C03563=1009.631,342.526,-157.819,170.244,53.143,160.444
C03564=1009.638,342.773,-157.854,170.253,53.138,160.444
C03565=1009.644,343.021,-157.889,170.261,53.133,160.445
C03566=1009.650,343.269,-157.924,170.269,53.128,160.445
C03567=1009.657,343.516,-157.959,170.277,53.124,160.446
C03568=1009.664,343.764,-157.994,170.285,53.119,160.447
C03569=1009.671,344.011,-158.030,170.294,53.114,160.447
C03570=1009.677,344.258,-158.064,170.303,53.109,160.448
C03571=1009.683,344.506,-158.100,170.311,53.104,160.448
C03572=1009.689,344.753,-158.135,170.319,53.099,160.449
C03573=1009.696,345.000,-158.170,170.327,53.095,160.450
C03574=1009.703,345.248,-158.205,170.335,53.090,160.450
C03575=1009.709,345.496,-158.241,170.344,53.085,160.450
C03576=1009.716,345.743,-158.276,170.352,53.081,160.451
C03577=1009.723,345.990,-158.311,170.360,53.076,160.452
C03578=1009.729,346.238,-158.347,170.368,53.071,160.452
C03579=1009.735,346.485,-158.382,170.376,53.067,160.453
C03580=1009.741,346.733,-158.418,170.385,53.062,160.453
C03581=1009.748,346.980,-158.453,170.394,53.057,160.454
C03582=1009.755,347.227,-158.490,170.402,53.052,160.454
C03583=1009.761,347.475,-158.525,170.411,53.048,160.455
C03584=1009.767,347.722,-158.561,170.419,53.043,160.456
C03585=1009.775,347.970,-158.597,170.427,53.039,160.456
C03586=1009.782,348.217,-158.632,170.435,53.034,160.457
C03587=1009.788,348.465,-158.668,170.444,53.030,160.458
C03588=1009.795,348.711,-158.703,170.452,53.025,160.458
C03589=1009.801,348.959,-158.739,170.462,53.020,160.459
C03590=1009.808,349.206,-158.775,170.470,53.016,160.459
C03591=1009.814,349.454,-158.811,170.478,53.011,160.460
C03592=1009.822,349.701,-158.847,170.486,53.006,160.461
C03593=1009.828,349.949,-158.883,170.495,53.002,160.461
C03594=1009.835,350.195,-158.919,170.503,52.998,160.462
C03595=1009.841,350.442,-158.955,170.512,52.993,160.463
C03596=1009.848,350.691,-158.991,170.521,52.989,160.463
C03597=1009.855,350.938,-159.027,170.530,52.984,160.464
C03598=1009.862,351.185,-159.062,170.538,52.979,160.465
C03599=1009.869,351.433,-159.099,170.546,52.975,160.465
C03600=1009.876,351.679,-159.135,170.555,52.971,160.466
C03601=1009.882,351.927,-159.171,170.564,52.966,160.467
C03602=1009.889,352.175,-159.207,170.572,52.962,160.467
C03603=1009.896,352.422,-159.243,170.581,52.957,160.468
C03604=1009.903,352.668,-159.279,170.590,52.953,160.469
C03605=1009.910,352.916,-159.316,170.598,52.949,160.469
C03606=1009.916,353.163,-159.352,170.608,52.944,160.470
C03607=1009.922,353.410,-159.389,170.616,52.940,160.471
C03608=1009.930,353.658,-159.425,170.624,52.935,160.471
C03609=1009.936,353.907,-159.462,170.633,52.931,160.472
C03610=1009.944,354.156,-159.498,170.642,52.927,160.473
C03611=1009.950,354.406,-159.536,170.651,52.922,160.474
C03612=1009.957,354.655,-159.572,170.659,52.918,160.474
C03613=1009.964,354.902,-159.609,170.669,52.914,160.475
C03614=1009.971,355.149,-159.645,170.678,52.909,160.476
C03615=1009.978,355.397,-159.681,170.686,52.905,160.477
C03616=1009.985,355.643,-159.719,170.695,52.901,160.477
C03617=1009.993,355.891,-159.755,170.704,52.896,160.478
C03618=1010.000,356.139,-159.792,170.713,52.893,160.479
C03619=1010.006,356.386,-159.828,170.722,52.889,160.480
C03620=1010.013,356.633,-159.866,170.731,52.884,160.481
C03621=1010.020,356.880,-159.901,170.740,52.880,160.481
C03622=1010.027,357.127,-159.938,170.748,52.876,160.482
C03623=1010.034,357.374,-159.976,170.757,52.872,160.483
C03624=1010.041,357.622,-160.012,170.767,52.867,160.484
C03625=1010.049,357.868,-160.049,170.775,52.863,160.485
C03626=1010.056,358.116,-160.086,170.784,52.859,160.485
C03627=1010.062,358.363,-160.123,170.794,52.855,160.486
C03628=1010.070,358.610,-160.161,170.803,52.851,160.487
C03629=1010.077,358.857,-160.197,170.811,52.847,160.488
C03630=1010.084,359.105,-160.235,170.821,52.843,160.489
C03631=1010.090,359.351,-160.272,170.830,52.838,160.489
C03632=1010.098,359.598,-160.310,170.839,52.835,160.490
C03633=1010.105,359.846,-160.347,170.848,52.830,160.491
C03634=1010.112,360.093,-160.384,170.857,52.827,160.492
C03635=1010.119,360.340,-160.422,170.866,52.823,160.493
C03636=1010.126,360.587,-160.459,170.876,52.819,160.494
C03637=1010.133,360.834,-160.496,170.884,52.814,160.495
C03638=1010.140,361.081,-160.534,170.893,52.811,160.495
C03639=1010.147,361.328,-160.571,170.903,52.806,160.496
C03640=1010.155,361.575,-160.609,170.912,52.803,160.497
C03641=1010.162,361.822,-160.646,170.922,52.799,160.498
C03642=1010.169,362.069,-160.684,170.930,52.795,160.499
C03643=1010.176,362.317,-160.721,170.939,52.791,160.500
C03644=1010.184,362.564,-160.759,170.949,52.787,160.501
C03645=1010.191,362.811,-160.796,170.958,52.783,160.502
C03646=1010.198,363.058,-160.834,170.968,52.779,160.503
C03647=1010.205,363.305,-160.872,170.977,52.775,160.504
C03648=1010.213,363.552,-160.910,170.987,52.771,160.505
C03649=1010.220,363.799,-160.947,170.995,52.767,160.505
C03650=1010.227,364.046,-160.985,171.005,52.763,160.506
C03651=1010.235,364.293,-161.022,171.014,52.760,160.507
C03652=1010.242,364.539,-161.061,171.023,52.756,160.508
C03653=1010.250,364.787,-161.098,171.033,52.752,160.509
C03654=1010.257,365.034,-161.136,171.042,52.749,160.510
C03655=1010.265,365.281,-161.174,171.052,52.745,160.511
C03656=1010.272,365.528,-161.212,171.061,52.741,160.512
C03657=1009.942,363.417,-161.243,170.962,52.829,160.514
C03658=1009.935,363.169,-161.206,170.952,52.833,160.513
C03659=1009.928,362.922,-161.168,170.943,52.836,160.512
C03660=1009.920,362.675,-161.131,170.934,52.840,160.511
C03661=1009.913,362.428,-161.093,170.924,52.844,160.510
C03662=1009.906,362.181,-161.056,170.915,52.848,160.509
C03663=1009.899,361.934,-161.018,170.905,52.852,160.508
C03664=1009.891,361.687,-160.981,170.897,52.856,160.508
C03665=1009.884,361.439,-160.943,170.887,52.860,160.507
C03666=1009.877,361.192,-160.906,170.878,52.864,160.506
C03667=1009.870,360.945,-160.868,170.869,52.868,160.505
C03668=1009.863,360.698,-160.831,170.859,52.872,160.504
C03669=1009.856,360.452,-160.793,170.851,52.876,160.503
C03670=1009.849,360.205,-160.756,170.842,52.880,160.502
C03671=1009.841,359.957,-160.718,170.832,52.884,160.501
C03672=1009.834,359.710,-160.682,170.823,52.888,160.501
C03673=1009.827,359.462,-160.644,170.814,52.892,160.500
C03674=1009.821,359.216,-160.607,170.805,52.896,160.499
C03675=1009.813,358.969,-160.569,170.796,52.900,160.498
C03676=1009.806,358.721,-160.532,170.786,52.904,160.497
C03677=1009.800,358.475,-160.495,170.778,52.908,160.496
C03678=1009.793,358.227,-160.459,170.769,52.913,160.496
C03679=1009.786,357.980,-160.421,170.759,52.917,160.495
C03680=1009.779,357.733,-160.385,170.751,52.921,160.494
C03681=1009.772,357.486,-160.347,170.742,52.925,160.493
C03682=1009.765,357.238,-160.310,170.733,52.929,160.492
C03683=1009.758,356.992,-160.274,170.723,52.933,160.491
C03684=1009.751,356.744,-160.237,170.715,52.937,160.491
C03685=1009.744,356.496,-160.200,170.706,52.942,160.490
C03686=1009.737,356.250,-160.163,170.697,52.946,160.489
C03687=1009.729,356.002,-160.127,170.688,52.950,160.488
C03688=1009.723,355.755,-160.090,170.679,52.954,160.487
C03689=1009.716,355.508,-160.053,170.670,52.959,160.487
C03690=1009.710,355.284,-160.021,170.662,52.962,160.486
C03691=1009.704,355.060,-159.988,170.655,52.966,160.485
C03692=1009.697,354.837,-159.954,170.646,52.970,160.485
C03693=1009.691,354.612,-159.921,170.639,52.974,160.484
C03694=1009.684,354.389,-159.888,170.630,52.978,160.483
C03695=1009.678,354.165,-159.855,170.623,52.982,160.483
C03696=1009.673,353.941,-159.822,170.615,52.986,160.482
C03697=1009.666,353.717,-159.789,170.606,52.990,160.481
C03698=1009.660,353.470,-159.753,170.598,52.994,160.481
C03699=1009.653,353.223,-159.716,170.589,52.999,160.480
C03700=1009.646,352.976,-159.680,170.581,53.003,160.479
C03701=1009.639,352.728,-159.644,170.571,53.008,160.478
C03702=1009.633,352.480,-159.608,170.563,53.012,160.478
C03703=1009.625,352.234,-159.572,170.554,53.016,160.477
C03704=1009.619,351.986,-159.535,170.546,53.020,160.476
C03705=1009.611,351.739,-159.499,170.537,53.025,160.476
C03706=1009.605,351.492,-159.464,170.528,53.030,160.475
C03707=1009.598,351.244,-159.427,170.519,53.034,160.474
C03708=1009.591,350.997,-159.391,170.511,53.038,160.474
C03709=1009.585,350.750,-159.356,170.503,53.043,160.473
C03710=1009.578,350.503,-159.319,170.494,53.047,160.472
C03711=1009.571,350.255,-159.284,170.485,53.052,160.472
C03712=1009.565,350.008,-159.247,170.477,53.057,160.471
C03713=1009.558,349.760,-159.212,170.468,53.061,160.470
C03714=1009.552,349.513,-159.176,170.459,53.065,160.470
C03715=1009.545,349.266,-159.141,170.451,53.070,160.469
C03716=1009.538,349.019,-159.104,170.443,53.074,160.468
C03717=1009.531,348.771,-159.069,170.434,53.079,160.468
C03718=1009.525,348.524,-159.032,170.425,53.084,160.467
C03719=1009.518,348.276,-158.997,170.417,53.089,160.467
C03720=1009.512,348.029,-158.961,170.409,53.093,160.466
C03721=1009.505,347.782,-158.926,170.400,53.098,160.465
C03722=1009.499,347.534,-158.890,170.392,53.102,160.465
C03723=1009.492,347.287,-158.855,170.384,53.107,160.464
C03724=1009.486,347.039,-158.819,170.374,53.111,160.463
C03725=1009.479,346.792,-158.783,170.366,53.116,160.463
C03726=1009.472,346.545,-158.748,170.358,53.121,160.462
C03727=1009.466,346.297,-158.712,170.349,53.125,160.462
C03728=1009.459,346.050,-158.677,170.341,53.130,160.461
C03729=1009.453,345.802,-158.641,170.333,53.135,160.461
C03730=1009.447,345.555,-158.606,170.325,53.139,160.460
C03731=1009.440,345.308,-158.571,170.317,53.144,160.459
C03732=1009.434,345.060,-158.535,170.309,53.149,160.459
C03733=1009.427,344.812,-158.500,170.300,53.154,160.458
C03734=1009.420,344.565,-158.465,170.291,53.159,160.457
C03735=1009.413,344.318,-158.430,170.283,53.163,160.457
C03736=1009.408,344.071,-158.395,170.275,53.168,160.456
C03737=1009.402,343.823,-158.360,170.267,53.173,160.456
C03738=1009.395,343.575,-158.325,170.259,53.178,160.455
C03739=1009.388,343.328,-158.290,170.250,53.183,160.455
C03740=1009.381,343.081,-158.255,170.242,53.187,160.454
C03741=1009.376,342.832,-158.220,170.234,53.192,160.454
C03742=1009.369,342.586,-158.185,170.226,53.197,160.453
C03743=1009.363,342.338,-158.150,170.218,53.202,160.453
C03744=1009.356,342.090,-158.115,170.209,53.207,160.452
C03745=1009.350,341.843,-158.080,170.201,53.212,160.452
C03746=1009.344,341.596,-158.045,170.193,53.216,160.451
C03747=1009.337,341.348,-158.011,170.185,53.221,160.451
C03748=1009.331,341.101,-157.975,170.177,53.226,160.450
C03749=1009.324,340.853,-157.941,170.169,53.231,160.450
C03750=1009.318,340.606,-157.906,170.161,53.236,160.449
C03751=1009.312,340.358,-157.871,170.153,53.241,160.449
C03752=1009.306,340.110,-157.836,170.145,53.246,160.448
C03753=1009.300,339.863,-157.802,170.137,53.251,160.448
C03754=1009.291,339.530,-157.756,170.125,53.259,160.447
C03755=1009.283,339.197,-157.709,170.114,53.265,160.446
C03756=1009.275,338.864,-157.662,170.104,53.271,160.446
C03757=1009.266,338.532,-157.616,170.093,53.278,160.445
C03758=1009.260,338.285,-157.581,170.085,53.284,160.445
C03759=1009.253,338.037,-157.547,170.077,53.289,160.444
C03760=1009.247,337.790,-157.513,170.069,53.293,160.444
C03761=1009.241,337.542,-157.478,170.061,53.298,160.443
C03762=1009.235,337.295,-157.444,170.053,53.304,160.443
C03763=1009.229,337.047,-157.410,170.045,53.309,160.442
C03764=1009.223,336.799,-157.376,170.037,53.314,160.442
C03765=1009.216,336.551,-157.342,170.030,53.319,160.442
C03766=1009.211,336.304,-157.307,170.021,53.324,160.441
C03767=1009.205,336.057,-157.273,170.014,53.330,160.441
C03768=1009.198,335.809,-157.239,170.006,53.335,160.440
C03769=1009.192,335.561,-157.205,169.998,53.339,160.440
C03770=1009.185,335.314,-157.171,169.990,53.345,160.440
C03771=1009.179,335.067,-157.137,169.983,53.350,160.439
C03772=1009.173,334.819,-157.103,169.975,53.355,160.439
C03773=1009.167,334.571,-157.069,169.967,53.360,160.438
C03774=1009.161,334.323,-157.035,169.960,53.366,160.438
C03775=1009.155,334.075,-157.001,169.951,53.370,160.438
C03776=1009.149,333.828,-156.967,169.944,53.376,160.437
C03777=1009.143,333.581,-156.933,169.936,53.382,160.437
C03778=1009.138,333.333,-156.899,169.928,53.386,160.436
C03779=1009.130,333.085,-156.866,169.920,53.392,160.436
C03780=1009.125,332.838,-156.832,169.912,53.397,160.436
C03781=1009.119,332.590,-156.798,169.905,53.403,160.435
C03782=1009.113,332.343,-156.764,169.897,53.408,160.435
C03783=1009.107,332.094,-156.730,169.889,53.413,160.435
C03784=1009.101,331.847,-156.696,169.881,53.419,160.434
C03785=1009.095,331.600,-156.662,169.875,53.424,160.434
C03786=1009.090,331.352,-156.629,169.867,53.429,160.434
C03787=1009.083,331.105,-156.596,169.859,53.434,160.433
C03788=1009.077,330.856,-156.562,169.851,53.440,160.433
C03789=1009.071,330.608,-156.528,169.844,53.445,160.433
C03790=1009.065,330.361,-156.495,169.836,53.450,160.432
C03791=1009.059,330.113,-156.462,169.828,53.456,160.432
C03792=1009.054,329.865,-156.428,169.820,53.461,160.432
C03793=1009.047,329.618,-156.395,169.813,53.467,160.431
C03794=1009.042,329.371,-156.362,169.805,53.473,160.431
C03795=1009.035,329.123,-156.329,169.797,53.478,160.431
C03796=1009.030,328.875,-156.295,169.791,53.483,160.430
C03797=1009.024,328.627,-156.262,169.783,53.488,160.430
C03798=1009.018,328.380,-156.229,169.775,53.494,160.430
C03799=1009.012,328.132,-156.195,169.767,53.499,160.429
C03800=1009.006,327.884,-156.162,169.760,53.505,160.429
C03801=1009.000,327.637,-156.129,169.752,53.511,160.429
C03802=1008.995,327.389,-156.096,169.744,53.516,160.428
C03803=1008.988,327.141,-156.063,169.737,53.522,160.428
C03804=1008.983,326.893,-156.030,169.730,53.527,160.428
C03805=1008.977,326.645,-155.996,169.723,53.532,160.428
C03806=1008.971,326.398,-155.964,169.715,53.538,160.427
C03807=1008.965,326.150,-155.930,169.707,53.544,160.427
C03808=1008.960,325.902,-155.897,169.700,53.549,160.427
C03809=1008.954,325.654,-155.864,169.692,53.555,160.426
C03810=1008.948,325.407,-155.831,169.686,53.561,160.427
C03811=1008.942,325.159,-155.798,169.678,53.566,160.426
C03812=1008.937,324.912,-155.765,169.671,53.572,160.426
C03813=1008.930,324.664,-155.733,169.663,53.577,160.426
C03814=1008.923,324.327,-155.689,169.653,53.585,160.425
C03815=1008.915,323.990,-155.644,169.643,53.593,160.425
C03816=1008.906,323.652,-155.601,169.633,53.600,160.425
C03817=1008.898,323.316,-155.556,169.623,53.609,160.424
C03818=1008.892,323.067,-155.524,169.615,53.614,160.424
C03819=1008.886,322.820,-155.491,169.608,53.620,160.424
C03820=1008.881,322.572,-155.459,169.601,53.626,160.424
C03821=1008.875,322.324,-155.426,169.593,53.632,160.423
C03822=1008.869,322.076,-155.394,169.585,53.637,160.423
C03823=1008.863,321.828,-155.361,169.579,53.643,160.423
C03824=1008.857,321.581,-155.330,169.572,53.649,160.423
C03825=1008.852,321.333,-155.296,169.564,53.654,160.423
C03826=1008.846,321.085,-155.264,169.557,53.661,160.422
C03827=1008.840,320.837,-155.233,169.549,53.666,160.422
C03828=1008.834,320.590,-155.200,169.542,53.672,160.422
C03829=1008.828,320.342,-155.168,169.535,53.678,160.422
C03830=1008.823,320.094,-155.136,169.528,53.683,160.422
C03831=1008.817,319.845,-155.104,169.521,53.690,160.422
C03832=1008.811,319.598,-155.071,169.513,53.695,160.421
C03833=1008.806,319.350,-155.039,169.506,53.701,160.421
C03834=1008.800,319.102,-155.007,169.498,53.707,160.421
C03835=1008.794,318.855,-154.976,169.492,53.713,160.421
C03836=1008.788,318.606,-154.944,169.484,53.719,160.420
C03837=1008.783,318.359,-154.911,169.477,53.725,160.420
C03838=1008.777,318.111,-154.879,169.470,53.731,160.420
C03839=1008.772,317.864,-154.847,169.462,53.737,160.420
C03840=1008.766,317.615,-154.815,169.456,53.743,160.420
C03841=1008.761,317.368,-154.783,169.449,53.748,160.420
C03842=1008.755,317.120,-154.751,169.441,53.755,160.420
C03843=1008.750,316.872,-154.719,169.434,53.761,160.420
C03844=1008.744,316.624,-154.687,169.428,53.766,160.419
C03845=1008.739,316.376,-154.655,169.420,53.772,160.419
C03846=1008.733,316.128,-154.623,169.413,53.778,160.419
C03847=1008.727,315.880,-154.592,169.406,53.784,160.419
C03848=1008.723,315.632,-154.559,169.398,53.790,160.419
C03849=1008.717,315.384,-154.527,169.392,53.796,160.419
C03850=1008.711,315.137,-154.496,169.385,53.802,160.419
C03851=1008.706,314.889,-154.464,169.378,53.808,160.418
C03852=1008.700,314.641,-154.432,169.370,53.815,160.418
C03853=1008.695,314.393,-154.401,169.364,53.820,160.418
C03854=1008.690,314.145,-154.369,169.357,53.826,160.418
C03855=1008.684,313.897,-154.337,169.349,53.832,160.418
C03856=1008.679,313.649,-154.305,169.342,53.839,160.418
C03857=1008.673,313.402,-154.273,169.336,53.845,160.418
C03858=1008.668,313.154,-154.242,169.328,53.850,160.418
C03859=1008.662,312.906,-154.210,169.321,53.857,160.417
C03860=1008.658,312.658,-154.178,169.315,53.862,160.417
C03861=1008.652,312.410,-154.146,169.308,53.869,160.417
C03862=1008.647,312.162,-154.116,169.301,53.875,160.417
C03863=1008.642,311.915,-154.084,169.294,53.881,160.417
C03864=1008.636,311.666,-154.052,169.288,53.887,160.417
C03865=1008.631,311.418,-154.021,169.280,53.894,160.417
C03866=1008.626,311.170,-153.989,169.273,53.899,160.417
C03867=1008.621,310.922,-153.958,169.266,53.905,160.417
C03868=1008.616,310.675,-153.926,169.259,53.911,160.417
C03869=1008.610,310.427,-153.894,169.252,53.918,160.417
C03870=1008.605,310.179,-153.863,169.245,53.924,160.417
C03871=1008.600,309.932,-153.832,169.239,53.930,160.417
C03872=1008.594,309.683,-153.800,169.232,53.936,160.416
C03873=1008.590,309.435,-153.768,169.225,53.943,160.416
C03874=1008.583,309.104,-153.727,169.216,53.951,160.417
C03875=1008.576,308.772,-153.685,169.207,53.959,160.416
C03876=1008.569,308.441,-153.643,169.197,53.967,160.416
C03877=1008.562,308.110,-153.602,169.189,53.976,160.416
C03878=1008.557,307.861,-153.571,169.182,53.982,160.416
C03879=1008.551,307.614,-153.540,169.175,53.989,160.416
C03880=1008.546,307.365,-153.509,169.168,53.994,160.416
C03881=1008.540,307.118,-153.479,169.162,54.001,160.416
C03882=1008.535,306.870,-153.448,169.155,54.008,160.416
C03883=1008.529,306.622,-153.418,169.147,54.014,160.416
C03884=1008.524,306.374,-153.387,169.141,54.020,160.416
C03885=1008.518,306.126,-153.357,169.134,54.026,160.416
C03886=1008.513,305.878,-153.326,169.127,54.033,160.416
C03887=1008.507,305.630,-153.295,169.120,54.040,160.416
C03888=1008.502,305.382,-153.264,169.114,54.046,160.416
C03889=1008.496,305.134,-153.234,169.107,54.053,160.416
C03890=1008.492,304.885,-153.204,169.100,54.059,160.416
C03891=1008.486,304.638,-153.174,169.093,54.065,160.416
C03892=1008.481,304.390,-153.143,169.087,54.071,160.416
C03893=1008.475,304.142,-153.112,169.080,54.078,160.416
C03894=1008.470,303.894,-153.081,169.073,54.085,160.416
C03895=1008.465,303.645,-153.052,169.067,54.090,160.416
C03896=1008.460,303.397,-153.021,169.060,54.098,160.416
C03897=1008.454,303.149,-152.991,169.053,54.104,160.416
C03898=1008.450,302.901,-152.961,169.047,54.111,160.416
C03899=1008.444,302.654,-152.930,169.040,54.117,160.416
C03900=1008.439,302.405,-152.899,169.033,54.123,160.416
C03901=1008.433,302.157,-152.870,169.027,54.130,160.416
C03902=1008.428,301.909,-152.839,169.020,54.136,160.416
C03903=1008.423,301.662,-152.809,169.014,54.143,160.416
C03904=1008.418,301.413,-152.779,169.007,54.149,160.416
C03905=1008.413,301.165,-152.748,169.001,54.156,160.416
C03906=1008.408,300.916,-152.718,168.994,54.162,160.416
C03907=1008.403,300.669,-152.688,168.987,54.169,160.416
C03908=1008.398,300.421,-152.658,168.981,54.175,160.416
C03909=1008.392,300.173,-152.627,168.974,54.182,160.417
C03910=1008.386,299.863,-152.590,168.966,54.190,160.416
C03911=1008.380,299.552,-152.552,168.957,54.199,160.417
C03912=1008.373,299.242,-152.514,168.949,54.207,160.417
C03913=1008.367,298.932,-152.477,168.941,54.215,160.417
C03914=1008.125,299.698,-152.935,168.938,54.244,160.423
C03915=1008.132,300.072,-152.980,168.949,54.235,160.423
C03916=1008.141,300.446,-153.026,168.958,54.225,160.423
C03917=1008.148,300.821,-153.072,168.968,54.215,160.423
C03918=1008.156,301.195,-153.117,168.978,54.206,160.423
C03919=1008.161,301.444,-153.147,168.985,54.198,160.423
C03920=1008.166,301.692,-153.178,168.991,54.193,160.423
C03921=1008.171,301.940,-153.207,168.998,54.186,160.423
C03922=1008.176,302.188,-153.238,169.005,54.179,160.423
C03923=1008.182,302.436,-153.268,169.011,54.173,160.423
C03924=1008.187,302.685,-153.299,169.018,54.166,160.422
C03925=1008.192,302.932,-153.329,169.025,54.160,160.423
C03926=1008.197,303.180,-153.359,169.031,54.154,160.423
C03927=1008.203,303.428,-153.389,169.038,54.147,160.422
C03928=1008.208,303.676,-153.420,169.045,54.141,160.423
C03929=1008.213,303.925,-153.450,169.051,54.135,160.423
C03930=1008.218,304.172,-153.480,169.058,54.128,160.423
C03931=1008.224,304.420,-153.511,169.065,54.121,160.423
C03932=1008.229,304.668,-153.542,169.072,54.115,160.423
C03933=1008.234,304.917,-153.571,169.078,54.109,160.423
C03934=1008.239,305.165,-153.602,169.085,54.103,160.423
C03935=1008.245,305.413,-153.633,169.092,54.096,160.423
C03936=1008.250,305.661,-153.664,169.098,54.090,160.423
C03937=1008.255,305.909,-153.695,169.105,54.083,160.423
C03938=1008.261,306.157,-153.724,169.112,54.077,160.423
C03939=1008.266,306.405,-153.755,169.120,54.071,160.423
C03940=1008.271,306.652,-153.785,169.125,54.064,160.423
C03941=1008.276,306.901,-153.816,169.132,54.058,160.423
C03942=1008.282,307.148,-153.846,169.139,54.051,160.423
C03943=1008.287,307.397,-153.877,169.146,54.045,160.423
C03944=1008.293,307.644,-153.908,169.153,54.039,160.423
C03945=1008.298,307.893,-153.939,169.160,54.033,160.423
C03946=1008.304,308.141,-153.969,169.167,54.026,160.423
C03947=1008.311,308.474,-154.011,169.175,54.018,160.423
C03948=1008.318,308.807,-154.053,169.185,54.010,160.423
C03949=1008.324,309.142,-154.095,169.194,54.001,160.423
C03950=1008.331,309.475,-154.137,169.203,53.993,160.423
C03951=1008.337,309.723,-154.169,169.210,53.987,160.423
C03952=1008.342,309.971,-154.200,169.217,53.980,160.424
C03953=1008.347,310.219,-154.232,169.223,53.974,160.424
C03954=1008.352,310.467,-154.263,169.230,53.968,160.424
C03955=1008.357,310.715,-154.295,169.238,53.962,160.424
C03956=1008.362,310.963,-154.326,169.245,53.956,160.424
C03957=1008.368,311.211,-154.357,169.251,53.950,160.424
C03958=1008.372,311.459,-154.389,169.259,53.944,160.424
C03959=1008.377,311.707,-154.421,169.266,53.938,160.424
C03960=1008.383,311.954,-154.452,169.272,53.932,160.424
C03961=1008.388,312.202,-154.483,169.279,53.925,160.424
C03962=1008.394,312.450,-154.515,169.287,53.920,160.425
C03963=1008.399,312.698,-154.547,169.294,53.913,160.425
C03964=1008.404,312.946,-154.578,169.300,53.908,160.425
C03965=1008.409,313.194,-154.610,169.307,53.901,160.425
C03966=1008.414,313.441,-154.642,169.314,53.895,160.425
C03967=1008.420,313.690,-154.674,169.321,53.890,160.425
C03968=1008.426,313.938,-154.705,169.328,53.883,160.425
C03969=1008.431,314.185,-154.736,169.335,53.877,160.425
C03970=1008.436,314.433,-154.768,169.342,53.871,160.425
C03971=1008.442,314.681,-154.801,169.349,53.866,160.426
C03972=1008.447,314.929,-154.832,169.356,53.859,160.426
C03973=1008.452,315.177,-154.863,169.363,53.853,160.426
C03974=1008.458,315.425,-154.895,169.371,53.847,160.426
C03975=1008.463,315.673,-154.927,169.377,53.841,160.426
C03976=1008.469,315.920,-154.959,169.384,53.835,160.426
C03977=1008.474,316.169,-154.991,169.392,53.830,160.427
C03978=1008.479,316.416,-155.023,169.399,53.823,160.427
C03979=1008.485,316.664,-155.054,169.406,53.818,160.427
C03980=1008.491,316.912,-155.087,169.413,53.812,160.427
C03981=1008.496,317.159,-155.118,169.420,53.805,160.427
C03982=1008.501,317.408,-155.151,169.428,53.800,160.427
C03983=1008.507,317.655,-155.182,169.435,53.794,160.427
C03984=1008.513,317.904,-155.214,169.441,53.788,160.428
C03985=1008.518,318.151,-155.246,169.449,53.782,160.428
C03986=1008.524,318.399,-155.278,169.456,53.776,160.428
C03987=1008.530,318.647,-155.310,169.463,53.770,160.428
C03988=1008.535,318.895,-155.342,169.470,53.765,160.428
C03989=1008.540,319.143,-155.374,169.477,53.759,160.428
C03990=1008.546,319.391,-155.407,169.485,53.753,160.429
C03991=1008.552,319.638,-155.439,169.492,53.747,160.429
C03992=1008.558,319.886,-155.471,169.500,53.741,160.429
C03993=1008.563,320.134,-155.502,169.507,53.735,160.429
C03994=1008.568,320.382,-155.535,169.513,53.730,160.429
C03995=1008.575,320.630,-155.568,169.521,53.724,160.430
C03996=1008.580,320.877,-155.599,169.528,53.718,160.430
C03997=1008.586,321.126,-155.631,169.536,53.712,160.430
C03998=1008.592,321.374,-155.663,169.543,53.706,160.430
C03999=1008.598,321.621,-155.696,169.550,53.701,160.430
C04000=1008.603,321.869,-155.728,169.557,53.695,160.431
C04001=1008.609,322.117,-155.761,169.565,53.689,160.431
C04002=1008.615,322.364,-155.793,169.572,53.683,160.431
C04003=1008.621,322.613,-155.825,169.580,53.677,160.431
C04004=1008.627,322.860,-155.857,169.587,53.672,160.432
C04005=1008.632,323.109,-155.890,169.595,53.666,160.432
C04006=1008.638,323.356,-155.922,169.601,53.660,160.432
C04007=1008.647,323.695,-155.966,169.612,53.653,160.433
C04008=1008.654,324.035,-156.011,169.623,53.645,160.433
C04009=1008.662,324.374,-156.056,169.632,53.637,160.433
C04010=1008.671,324.713,-156.100,169.642,53.629,160.434
C04011=1008.677,324.961,-156.133,169.650,53.624,160.434
C04012=1008.682,325.209,-156.165,169.658,53.618,160.434
C04013=1008.687,325.457,-156.198,169.665,53.613,160.434
C04014=1008.693,325.704,-156.231,169.671,53.607,160.434
C04015=1008.699,325.952,-156.264,169.679,53.601,160.435
C04016=1008.705,326.200,-156.298,169.687,53.596,160.435
C04017=1008.711,326.448,-156.330,169.694,53.590,160.435
C04018=1008.716,326.695,-156.364,169.702,53.584,160.436
C04019=1008.723,326.943,-156.396,169.710,53.579,160.436
C04020=1008.728,327.191,-156.430,169.716,53.574,160.436
C04021=1008.734,327.439,-156.463,169.724,53.569,160.437
C04022=1008.740,327.686,-156.496,169.732,53.563,160.437
C04023=1008.745,327.934,-156.529,169.740,53.558,160.437
C04024=1008.751,328.182,-156.562,169.747,53.552,160.438
C04025=1008.757,328.429,-156.595,169.755,53.546,160.438
C04026=1008.762,328.677,-156.628,169.763,53.541,160.438
C04027=1008.769,328.924,-156.662,169.770,53.535,160.438
C04028=1008.775,329.173,-156.695,169.777,53.530,160.439
C04029=1008.781,329.421,-156.729,169.784,53.524,160.439
C04030=1008.787,329.668,-156.761,169.793,53.520,160.440
C04031=1008.793,329.916,-156.795,169.800,53.514,160.440
C04032=1008.798,330.163,-156.829,169.808,53.508,160.440
C04033=1008.805,330.411,-156.862,169.815,53.503,160.440
C04034=1008.810,330.659,-156.895,169.823,53.497,160.441
C04035=1008.816,330.906,-156.929,169.831,53.492,160.441
C04036=1008.822,331.154,-156.962,169.839,53.487,160.442
C04037=1008.828,331.402,-156.995,169.846,53.481,160.442
C04038=1008.834,331.650,-157.029,169.855,53.476,160.442
C04039=1008.840,331.898,-157.063,169.861,53.471,160.443
C04040=1008.846,332.145,-157.097,169.869,53.465,160.443
C04041=1008.851,332.393,-157.130,169.877,53.461,160.443
C04042=1008.858,332.640,-157.164,169.885,53.455,160.444
C04043=1008.864,332.887,-157.198,169.893,53.450,160.444
C04044=1008.870,333.136,-157.231,169.900,53.444,160.444
C04045=1008.876,333.383,-157.265,169.908,53.439,160.445
C04046=1008.882,333.630,-157.300,169.916,53.434,160.445
C04047=1008.887,333.878,-157.333,169.924,53.428,160.446
C04048=1008.894,334.126,-157.367,169.932,53.423,160.446
C04049=1008.900,334.373,-157.401,169.939,53.418,160.446
C04050=1008.905,334.621,-157.435,169.948,53.413,160.447
C04051=1008.912,334.869,-157.468,169.955,53.407,160.447
C04052=1008.918,335.116,-157.503,169.963,53.403,160.448
C04053=1008.924,335.363,-157.537,169.971,53.397,160.448
C04054=1008.931,335.611,-157.571,169.979,53.392,160.449
C04055=1008.936,335.859,-157.605,169.986,53.388,160.449
C04056=1008.943,336.107,-157.639,169.994,53.382,160.449
C04057=1008.948,336.355,-157.673,170.002,53.377,160.450
C04058=1008.954,336.602,-157.707,170.009,53.371,160.450
C04059=1008.961,336.850,-157.741,170.018,53.367,160.451
C04060=1008.967,337.097,-157.775,170.026,53.362,160.451
C04061=1008.974,337.345,-157.809,170.033,53.356,160.451
C04062=1008.980,337.592,-157.843,170.041,53.351,160.452
C04063=1008.986,337.840,-157.878,170.049,53.346,160.452
C04064=1008.992,338.087,-157.912,170.058,53.341,160.453
C04065=1008.998,338.335,-157.947,170.066,53.337,160.453
C04066=1009.004,338.582,-157.981,170.073,53.331,160.454
C04067=1009.013,338.917,-158.028,170.084,53.324,160.454
C04068=1009.021,339.252,-158.075,170.096,53.317,160.455
C04069=1009.029,339.588,-158.121,170.107,53.311,160.456
C04070=1009.038,339.922,-158.168,170.117,53.304,160.457
C04071=1009.044,340.169,-158.203,170.125,53.299,160.457
C04072=1009.050,340.418,-158.238,170.134,53.294,160.458
C04073=1009.056,340.664,-158.273,170.141,53.289,160.458
C04074=1009.063,340.912,-158.307,170.149,53.284,160.458
C04075=1009.069,341.160,-158.342,170.157,53.279,160.459
C04076=1009.075,341.407,-158.376,170.165,53.274,160.459
C04077=1009.082,341.654,-158.411,170.174,53.269,160.460
C04078=1009.088,341.903,-158.446,170.182,53.264,160.460
C04079=1009.094,342.149,-158.481,170.190,53.259,160.461
C04080=1009.100,342.397,-158.516,170.198,53.255,160.462
C04081=1009.107,342.645,-158.551,170.206,53.250,160.462
C04082=1009.113,342.892,-158.587,170.216,53.245,160.463
C04083=1009.120,343.140,-158.621,170.224,53.240,160.463
C04084=1009.126,343.387,-158.656,170.232,53.235,160.464
C04085=1009.133,343.634,-158.691,170.240,53.230,160.464
C04086=1009.139,343.882,-158.725,170.248,53.226,160.465
C04087=1009.145,344.130,-158.761,170.256,53.221,160.466
C04088=1009.152,344.377,-158.796,170.265,53.216,160.466
C04089=1009.159,344.625,-158.831,170.273,53.211,160.467
C04090=1009.165,344.871,-158.866,170.281,53.207,160.467
C04091=1009.171,345.119,-158.902,170.289,53.202,160.468
C04092=1009.177,345.367,-158.936,170.297,53.197,160.468
C04093=1009.184,345.614,-158.971,170.307,53.192,160.469
C04094=1009.190,345.862,-159.007,170.315,53.187,160.469
C04095=1009.197,346.109,-159.043,170.323,53.183,160.470
C04096=1009.204,346.356,-159.078,170.331,53.178,160.471
C04097=1009.210,346.604,-159.114,170.339,53.173,160.471
C04098=1009.217,346.851,-159.149,170.348,53.169,160.472
C04099=1009.223,347.099,-159.185,170.356,53.164,160.472
C04100=1009.230,347.346,-159.220,170.365,53.160,160.473
C04101=1009.236,347.594,-159.256,170.373,53.155,160.474
C04102=1009.243,347.841,-159.291,170.382,53.150,160.475
C04103=1009.249,348.088,-159.327,170.390,53.146,160.475
C04104=1009.255,348.336,-159.362,170.399,53.141,160.476
C04105=1009.262,348.583,-159.399,170.407,53.136,160.476
C04106=1009.269,348.830,-159.434,170.415,53.132,160.477
C04107=1009.275,349.078,-159.470,170.424,53.127,160.477
C04108=1009.282,349.325,-159.505,170.432,53.123,160.478
C04109=1009.288,349.573,-159.541,170.442,53.119,160.479
C04110=1009.295,349.820,-159.577,170.450,53.114,160.480
C04111=1009.302,350.067,-159.612,170.458,53.109,160.480
C04112=1009.308,350.314,-159.649,170.467,53.105,160.481
C04113=1009.315,350.562,-159.684,170.475,53.100,160.481
C04114=1009.322,350.809,-159.721,170.485,53.096,160.482
C04115=1009.329,351.057,-159.756,170.493,53.091,160.483
C04116=1009.335,351.304,-159.792,170.501,53.087,160.484
C04117=1009.342,351.551,-159.828,170.510,53.082,160.484
C04118=1009.349,351.799,-159.864,170.518,53.078,160.485
C04119=1009.356,352.046,-159.900,170.528,53.074,160.486
C04120=1009.362,352.293,-159.936,170.536,53.069,160.487
C04121=1009.369,352.540,-159.972,170.544,53.064,160.487
C04122=1009.376,352.788,-160.009,170.553,53.060,160.488
C04123=1009.382,353.035,-160.045,170.563,53.056,160.489
C04124=1009.389,353.282,-160.082,170.571,53.051,160.489
C04125=1009.396,353.529,-160.118,170.580,53.047,160.490
C04126=1009.403,353.776,-160.154,170.588,53.043,160.491
C04127=1009.414,354.175,-160.212,170.602,53.036,160.492
C04128=1009.425,354.573,-160.272,170.617,53.029,160.493
C04129=1009.436,354.971,-160.329,170.631,53.022,160.494
C04130=1009.447,355.369,-160.388,170.645,53.015,160.496
C04131=1009.454,355.616,-160.425,170.654,53.011,160.496
C04132=1009.461,355.864,-160.462,170.664,53.006,160.497
C04133=1009.468,356.110,-160.498,170.672,53.002,160.498
C04134=1009.475,356.357,-160.535,170.681,52.998,160.499
C04135=1009.481,356.604,-160.571,170.691,52.994,160.500
C04136=1009.488,356.852,-160.608,170.699,52.990,160.500
C04137=1009.496,357.098,-160.645,170.708,52.986,160.501
C04138=1009.503,357.346,-160.682,170.717,52.981,160.502
C04139=1009.510,357.594,-160.718,170.726,52.977,160.503
C04140=1009.516,357.840,-160.756,170.735,52.973,160.504
C04141=1009.523,358.088,-160.792,170.744,52.968,160.505
C04142=1009.530,358.335,-160.830,170.753,52.964,160.505
C04143=1009.537,358.582,-160.866,170.762,52.961,160.506
C04144=1009.544,358.829,-160.904,170.771,52.956,160.507
C04145=1009.551,359.077,-160.941,170.780,52.953,160.508
C04146=1009.558,359.324,-160.978,170.789,52.948,160.509
C04147=1009.565,359.571,-161.015,170.799,52.944,160.510
C04148=1009.572,359.818,-161.053,170.807,52.940,160.510
C04149=1009.579,360.064,-161.090,170.817,52.937,160.511
C04150=1009.586,360.312,-161.127,170.826,52.932,160.512
C04151=1009.593,360.559,-161.164,170.835,52.928,160.513
C04152=1009.600,360.806,-161.202,170.845,52.924,160.514
C04153=1009.607,361.053,-161.239,170.854,52.920,160.515
C04154=1009.614,361.300,-161.277,170.862,52.916,160.516
C04155=1009.289,359.188,-161.313,170.765,53.003,160.517
C04156=1009.283,358.942,-161.276,170.756,53.007,160.517
C04157=1009.275,358.695,-161.238,170.746,53.011,160.516
C04158=1009.269,358.447,-161.201,170.738,53.016,160.515
C04159=1009.262,358.201,-161.164,170.729,53.019,160.514
C04160=1009.255,357.953,-161.127,170.719,53.024,160.513
C04161=1009.248,357.707,-161.091,170.711,53.028,160.512
C04162=1009.241,357.459,-161.054,170.702,53.032,160.511
C04163=1009.234,357.211,-161.017,170.692,53.036,160.511
C04164=1009.227,356.964,-160.981,170.684,53.040,160.510
C04165=1009.219,356.717,-160.944,170.675,53.045,160.509
C04166=1009.213,356.470,-160.907,170.665,53.049,160.508
C04167=1009.206,356.223,-160.871,170.656,53.053,160.507
C04168=1009.200,355.976,-160.834,170.648,53.057,160.507
C04169=1009.192,355.728,-160.798,170.638,53.062,160.506
C04170=1009.185,355.482,-160.761,170.630,53.066,160.505
C04171=1009.179,355.234,-160.724,170.621,53.070,160.504
C04172=1009.169,354.885,-160.674,170.609,53.076,160.503
C04173=1009.159,354.536,-160.622,170.595,53.082,160.502
C04174=1009.149,354.185,-160.570,170.583,53.089,160.501
C04175=1009.140,353.837,-160.519,170.571,53.095,160.500
C04176=1009.133,353.588,-160.482,170.562,53.099,160.499
C04177=1009.126,353.341,-160.447,170.553,53.103,160.498
C04178=1009.120,353.094,-160.410,170.544,53.108,160.498
C04179=1009.113,352.847,-160.373,170.535,53.112,160.497
C04180=1009.106,352.600,-160.337,170.527,53.116,160.496
C04181=1009.100,352.353,-160.301,170.518,53.120,160.495
C04182=1009.094,352.105,-160.265,170.510,53.125,160.495
C04183=1009.086,351.858,-160.229,170.501,53.130,160.494
C04184=1009.079,351.611,-160.193,170.492,53.134,160.493
C04185=1009.073,351.363,-160.158,170.484,53.138,160.493
C04186=1009.066,351.117,-160.122,170.475,53.143,160.492
C04187=1009.059,350.868,-160.086,170.466,53.148,160.491
C04188=1009.052,350.621,-160.050,170.457,53.152,160.491
C04189=1009.046,350.374,-160.014,170.449,53.156,160.490
C04190=1009.039,350.127,-159.978,170.440,53.161,160.489
C04191=1009.033,349.879,-159.942,170.432,53.165,160.489
C04192=1009.026,349.632,-159.907,170.423,53.170,160.488
C04193=1009.019,349.384,-159.870,170.414,53.174,160.487
C04194=1009.012,349.137,-159.835,170.406,53.179,160.487
C04195=1009.006,348.890,-159.799,170.397,53.183,160.486
C04196=1008.999,348.642,-159.764,170.389,53.188,160.485
C04197=1008.993,348.395,-159.728,170.381,53.193,160.485
C04198=1008.987,348.147,-159.693,170.372,53.198,160.484
C04199=1008.980,347.900,-159.656,170.363,53.202,160.483
C04200=1008.973,347.653,-159.621,170.355,53.207,160.483
C04201=1008.967,347.405,-159.586,170.346,53.211,160.482
C04202=1008.961,347.158,-159.550,170.338,53.216,160.481
C04203=1008.955,346.910,-159.515,170.330,53.220,160.481
C04204=1008.948,346.663,-159.480,170.322,53.225,160.480
C04205=1008.941,346.416,-159.443,170.312,53.230,160.479
C04206=1008.935,346.168,-159.408,170.304,53.235,160.479
C04207=1008.928,345.921,-159.373,170.296,53.239,160.478
C04208=1008.922,345.673,-159.337,170.287,53.244,160.478
C04209=1008.916,345.427,-159.302,170.279,53.249,160.477
C04210=1008.909,345.179,-159.268,170.271,53.253,160.476
C04211=1008.903,344.931,-159.232,170.263,53.258,160.476
C04212=1008.896,344.684,-159.197,170.255,53.263,160.475
C04213=1008.890,344.436,-159.162,170.246,53.268,160.475
C04214=1008.883,344.189,-159.127,170.237,53.272,160.474
C04215=1008.877,343.941,-159.092,170.229,53.277,160.473
C04216=1008.871,343.694,-159.057,170.221,53.282,160.473
C04217=1008.864,343.447,-159.022,170.213,53.287,160.472
C04218=1008.858,343.199,-158.987,170.205,53.292,160.472
C04219=1008.851,342.951,-158.952,170.196,53.296,160.471
C04220=1008.846,342.704,-158.917,170.188,53.301,160.471
C04221=1008.839,342.456,-158.883,170.180,53.306,160.470
C04222=1008.832,342.209,-158.847,170.172,53.311,160.470
C04223=1008.826,341.961,-158.813,170.164,53.316,160.469
C04224=1008.821,341.714,-158.778,170.156,53.321,160.469
C04225=1008.814,341.466,-158.743,170.147,53.326,160.468
C04226=1008.808,341.219,-158.708,170.139,53.330,160.468
C04227=1008.801,340.971,-158.674,170.131,53.335,160.467
C04228=1008.795,340.724,-158.639,170.123,53.340,160.467
C04229=1008.789,340.477,-158.605,170.115,53.345,160.466
C04230=1008.783,340.229,-158.569,170.107,53.350,160.466
C04231=1008.776,339.981,-158.535,170.099,53.355,160.465
C04232=1008.768,339.644,-158.488,170.087,53.362,160.464
C04233=1008.760,339.307,-158.441,170.077,53.369,160.464
C04234=1008.751,338.969,-158.393,170.066,53.376,160.463
C04235=1008.743,338.632,-158.347,170.054,53.382,160.462
C04236=1008.737,338.385,-158.313,170.046,53.388,160.462
C04237=1008.730,338.137,-158.278,170.038,53.393,160.461
C04238=1008.725,337.890,-158.244,170.030,53.398,160.461
C04239=1008.718,337.642,-158.209,170.023,53.402,160.460
C04240=1008.712,337.395,-158.175,170.015,53.407,160.460
C04241=1008.706,337.147,-158.141,170.007,53.413,160.460
C04242=1008.700,336.900,-158.107,169.999,53.417,160.459
C04243=1008.694,336.652,-158.073,169.991,53.422,160.458
C04244=1008.688,336.404,-158.038,169.983,53.428,160.458
C04245=1008.682,336.156,-158.005,169.975,53.433,160.458
C04246=1008.676,335.908,-157.971,169.967,53.438,160.457
C04247=1008.669,335.661,-157.937,169.959,53.443,160.457
C04248=1008.663,335.414,-157.903,169.951,53.448,160.456
C04249=1008.657,335.166,-157.869,169.944,53.454,160.456
C04250=1008.651,334.918,-157.835,169.936,53.459,160.455
C04251=1008.645,334.671,-157.801,169.928,53.464,160.455
C04252=1008.639,334.423,-157.767,169.920,53.469,160.455
C04253=1008.633,334.176,-157.733,169.912,53.474,160.454
C04254=1008.627,333.928,-157.699,169.904,53.480,160.454
C04255=1008.621,333.680,-157.665,169.896,53.485,160.453
C04256=1008.614,333.433,-157.632,169.888,53.490,160.453
C04257=1008.609,333.185,-157.598,169.880,53.495,160.452
C04258=1008.603,332.938,-157.564,169.873,53.501,160.452
C04259=1008.597,332.690,-157.531,169.865,53.506,160.452
C04260=1008.591,332.442,-157.497,169.857,53.511,160.451
C04261=1008.586,332.195,-157.463,169.849,53.517,160.451
C04262=1008.579,331.947,-157.429,169.842,53.521,160.451
C04263=1008.574,331.699,-157.396,169.835,53.527,160.450
C04264=1008.568,331.451,-157.362,169.826,53.532,160.450
C04265=1008.562,331.204,-157.329,169.819,53.537,160.449
C04266=1008.556,330.956,-157.295,169.811,53.543,160.449
C04267=1008.550,330.709,-157.261,169.803,53.548,160.449
C04268=1008.544,330.461,-157.229,169.795,53.554,160.448
C04269=1008.538,330.213,-157.195,169.788,53.559,160.448
C04270=1008.533,329.966,-157.161,169.780,53.565,160.448
C04271=1008.526,329.718,-157.129,169.772,53.570,160.447
C04272=1008.521,329.470,-157.095,169.765,53.575,160.447
C04273=1008.515,329.222,-157.062,169.758,53.580,160.447
C04274=1008.509,328.975,-157.029,169.750,53.586,160.446
C04275=1008.503,328.727,-156.996,169.743,53.592,160.446
C04276=1008.497,328.479,-156.963,169.734,53.597,160.446
C04277=1008.491,328.231,-156.930,169.727,53.602,160.445
C04278=1008.486,327.984,-156.896,169.719,53.608,160.445
C04279=1008.479,327.737,-156.863,169.712,53.613,160.445
C04280=1008.474,327.489,-156.830,169.704,53.619,160.444
C04281=1008.468,327.241,-156.796,169.697,53.624,160.444
C04282=1008.462,326.992,-156.764,169.690,53.630,160.444
C04283=1008.457,326.745,-156.731,169.682,53.635,160.443
C04284=1008.450,326.497,-156.698,169.674,53.641,160.443
C04285=1008.445,326.249,-156.665,169.667,53.647,160.443
C04286=1008.440,326.002,-156.632,169.659,53.652,160.443
C04287=1008.434,325.754,-156.599,169.653,53.657,160.442
C04288=1008.428,325.506,-156.566,169.645,53.663,160.442
C04289=1008.422,325.258,-156.532,169.637,53.669,160.442
C04290=1008.416,325.010,-156.500,169.630,53.674,160.441
C04291=1008.412,324.763,-156.467,169.622,53.680,160.441
C04292=1008.403,324.421,-156.423,169.612,53.687,160.441
C04293=1008.395,324.080,-156.378,169.602,53.695,160.440
C04294=1008.387,323.738,-156.334,169.592,53.703,160.440
C04295=1008.379,323.396,-156.289,169.581,53.711,160.440
C04296=1008.373,323.148,-156.256,169.573,53.716,160.439
C04297=1008.367,322.900,-156.224,169.566,53.722,160.439
C04298=1008.361,322.653,-156.192,169.559,53.728,160.439
C04299=1008.355,322.405,-156.160,169.552,53.734,160.439
C04300=1008.349,322.157,-156.128,169.544,53.739,160.438
C04301=1008.344,321.910,-156.095,169.536,53.745,160.438
C04302=1008.338,321.661,-156.063,169.529,53.751,160.438
C04303=1008.332,321.413,-156.031,169.523,53.756,160.438
C04304=1008.327,321.166,-155.998,169.515,53.762,160.437
C04305=1008.321,320.918,-155.966,169.508,53.768,160.437
C04306=1008.315,320.670,-155.934,169.500,53.774,160.437
C04307=1008.310,320.422,-155.902,169.493,53.779,160.437
C04308=1008.304,320.174,-155.870,169.486,53.785,160.437
C04309=1008.298,319.927,-155.837,169.479,53.791,160.436
C04310=1008.292,319.679,-155.805,169.471,53.797,160.436
C04311=1008.287,319.431,-155.774,169.464,53.803,160.436
C04312=1008.282,319.183,-155.741,169.456,53.808,160.436
C04313=1008.276,318.935,-155.709,169.450,53.814,160.436
C04314=1008.270,318.687,-155.677,169.443,53.820,160.435
C04315=1008.265,318.439,-155.646,169.435,53.826,160.435
C04316=1008.259,318.191,-155.614,169.428,53.832,160.435
C04317=1008.253,317.944,-155.582,169.420,53.838,160.435
C04318=1008.248,317.695,-155.549,169.414,53.843,160.435
C04319=1008.243,317.448,-155.518,169.406,53.849,160.434
C04320=1008.237,317.200,-155.486,169.399,53.855,160.434
C04321=1008.231,316.952,-155.454,169.392,53.861,160.434
C04322=1008.226,316.704,-155.422,169.385,53.867,160.434
C04323=1008.220,316.456,-155.390,169.378,53.872,160.434
C04324=1008.215,316.208,-155.358,169.371,53.879,160.433
C04325=1008.210,315.961,-155.327,169.363,53.885,160.433
C04326=1008.204,315.713,-155.294,169.357,53.890,160.433
C04327=1008.199,315.465,-155.263,169.350,53.897,160.433
C04328=1008.194,315.217,-155.232,169.342,53.902,160.433
C04329=1008.188,314.970,-155.200,169.335,53.909,160.433
C04330=1008.183,314.721,-155.168,169.329,53.915,160.433
C04331=1008.178,314.474,-155.136,169.321,53.920,160.432
C04332=1008.173,314.225,-155.105,169.314,53.926,160.432
C04333=1008.167,313.978,-155.073,169.307,53.933,160.432
C04334=1008.161,313.730,-155.041,169.300,53.938,160.432
C04335=1008.156,313.482,-155.010,169.293,53.944,160.432
C04336=1008.151,313.234,-154.978,169.286,53.951,160.432
C04337=1008.146,312.986,-154.946,169.279,53.956,160.431
C04338=1008.141,312.739,-154.915,169.272,53.962,160.431
C04339=1008.135,312.490,-154.883,169.265,53.969,160.431
C04340=1008.130,312.242,-154.852,169.258,53.975,160.431
C04341=1008.125,311.994,-154.821,169.251,53.980,160.431
C04342=1008.120,311.746,-154.789,169.244,53.986,160.431
C04343=1008.115,311.498,-154.758,169.237,53.993,160.431
C04344=1008.109,311.251,-154.726,169.231,53.999,160.431
C04345=1008.104,311.003,-154.695,169.224,54.005,160.431
C04346=1008.099,310.755,-154.663,169.216,54.011,160.431
C04347=1008.094,310.507,-154.632,169.210,54.017,160.430
C04348=1008.089,310.259,-154.600,169.203,54.023,160.430
C04349=1008.084,310.011,-154.569,169.195,54.029,160.430
C04350=1008.079,309.764,-154.538,169.189,54.035,160.430
C04351=1008.074,309.515,-154.507,169.182,54.041,160.430
C04352=1008.066,309.180,-154.464,169.172,54.050,160.430
C04353=1008.060,308.843,-154.422,169.163,54.058,160.430
C04354=1008.053,308.508,-154.379,169.155,54.066,160.430
C04355=1008.046,308.172,-154.337,169.145,54.075,160.429
C04356=1008.040,307.924,-154.306,169.138,54.081,160.429
C04357=1008.036,307.675,-154.276,169.131,54.087,160.429
C04358=1008.030,307.427,-154.246,169.124,54.093,160.429
C04359=1008.025,307.179,-154.215,169.117,54.100,160.429
C04360=1008.019,306.932,-154.184,169.110,54.106,160.429
C04361=1008.014,306.683,-154.154,169.104,54.112,160.429
C04362=1008.008,306.436,-154.123,169.097,54.119,160.429
C04363=1008.003,306.187,-154.092,169.090,54.125,160.429
C04364=1007.997,305.939,-154.063,169.083,54.132,160.429
C04365=1007.992,305.691,-154.032,169.077,54.137,160.429
C04366=1007.987,305.444,-154.002,169.070,54.144,160.429
C04367=1007.982,305.196,-153.971,169.063,54.150,160.429
C04368=1007.977,304.947,-153.940,169.056,54.156,160.429
C04369=1007.971,304.699,-153.910,169.050,54.163,160.429
C04370=1007.966,304.451,-153.879,169.043,54.169,160.429
C04371=1007.961,304.203,-153.849,169.036,54.175,160.429
C04372=1007.956,303.955,-153.819,169.029,54.182,160.429
C04373=1007.951,303.707,-153.789,169.023,54.189,160.429
C04374=1007.945,303.459,-153.758,169.017,54.195,160.429
C04375=1007.940,303.211,-153.728,169.009,54.201,160.429
C04376=1007.935,302.963,-153.697,169.002,54.207,160.429
C04377=1007.930,302.715,-153.668,168.997,54.214,160.429
C04378=1007.925,302.467,-153.637,168.989,54.220,160.429
C04379=1007.919,302.218,-153.607,168.982,54.227,160.429
C04380=1007.915,301.996,-153.580,168.976,54.233,160.429
C04381=1007.911,301.772,-153.552,168.971,54.238,160.429
C04382=1007.906,301.549,-153.525,168.965,54.244,160.429
C04383=1007.901,301.326,-153.498,168.959,54.250,160.429
C04384=1007.897,301.103,-153.472,168.953,54.256,160.429
C04385=1007.892,300.880,-153.444,168.947,54.261,160.429
C04386=1007.888,300.657,-153.417,168.941,54.267,160.429
C04387=1007.883,300.433,-153.390,168.935,54.273,160.429
C04388=1007.641,301.143,-153.842,168.932,54.301,160.434
C04389=1007.646,301.419,-153.875,168.939,54.293,160.434
C04390=1007.652,301.696,-153.909,168.946,54.286,160.434
C04391=1007.657,301.973,-153.942,168.954,54.279,160.434
C04392=1007.663,302.250,-153.976,168.961,54.272,160.434
C04393=1007.668,302.497,-154.006,168.968,54.266,160.434
C04394=1007.673,302.746,-154.036,168.975,54.259,160.434
C04395=1007.679,302.993,-154.067,168.981,54.253,160.434
C04396=1007.684,303.242,-154.097,168.988,54.247,160.434
C04397=1007.689,303.489,-154.127,168.995,54.240,160.434
C04398=1007.694,303.737,-154.158,169.001,54.234,160.434
C04399=1007.699,303.986,-154.187,169.008,54.227,160.434
C04400=1007.704,304.234,-154.218,169.015,54.221,160.434
C04401=1007.710,304.481,-154.248,169.021,54.215,160.434
C04402=1007.714,304.730,-154.279,169.028,54.209,160.435
C04403=1007.720,304.978,-154.309,169.035,54.202,160.435
C04404=1007.725,305.227,-154.339,169.041,54.196,160.435
C04405=1007.731,305.474,-154.369,169.049,54.190,160.435
C04406=1007.735,305.722,-154.400,169.056,54.184,160.435
C04407=1007.741,305.970,-154.430,169.062,54.178,160.435
C04408=1007.746,306.218,-154.461,169.069,54.171,160.435
C04409=1007.752,306.466,-154.491,169.076,54.164,160.435
C04410=1007.757,306.714,-154.522,169.082,54.158,160.435
C04411=1007.762,306.962,-154.552,169.089,54.152,160.435
C04412=1007.768,307.210,-154.583,169.096,54.146,160.435
C04413=1007.772,307.459,-154.613,169.102,54.140,160.435
C04414=1007.778,307.707,-154.644,169.109,54.133,160.435
C04415=1007.783,307.955,-154.675,169.117,54.127,160.435
C04416=1007.789,308.203,-154.705,169.124,54.121,160.435
C04417=1007.796,308.541,-154.747,169.132,54.113,160.436
C04418=1007.802,308.878,-154.790,169.142,54.105,160.436
C04419=1007.810,309.217,-154.833,169.152,54.096,160.436
C04420=1007.816,309.555,-154.875,169.161,54.087,160.436
C04421=1007.821,309.803,-154.907,169.168,54.082,160.436
C04422=1007.826,310.051,-154.938,169.175,54.076,160.436
C04423=1007.831,310.299,-154.970,169.182,54.070,160.437
C04424=1007.836,310.547,-155.001,169.188,54.064,160.436
C04425=1007.841,310.795,-155.031,169.195,54.057,160.437
C04426=1007.847,311.042,-155.063,169.203,54.052,160.437
C04427=1007.851,311.291,-155.095,169.209,54.046,160.437
C04428=1007.856,311.538,-155.126,169.216,54.039,160.437
C04429=1007.861,311.787,-155.157,169.223,54.033,160.437
C04430=1007.867,312.034,-155.189,169.230,54.028,160.437
C04431=1007.873,312.283,-155.220,169.237,54.021,160.437
C04432=1007.878,312.530,-155.252,169.244,54.015,160.438
C04433=1007.883,312.778,-155.284,169.250,54.009,160.438
C04434=1007.888,313.026,-155.315,169.258,54.004,160.438
C04435=1007.893,313.274,-155.347,169.265,53.997,160.438
C04436=1007.898,313.522,-155.378,169.273,53.992,160.438
C04437=1007.904,313.770,-155.409,169.279,53.986,160.438
C04438=1007.909,314.017,-155.441,169.286,53.979,160.438
C04439=1007.914,314.266,-155.473,169.294,53.974,160.439
C04440=1007.919,314.514,-155.505,169.300,53.968,160.439
C04441=1007.925,314.761,-155.536,169.307,53.961,160.439
C04442=1007.930,315.009,-155.568,169.315,53.956,160.439
C04443=1007.936,315.258,-155.599,169.322,53.949,160.439
C04444=1007.941,315.505,-155.631,169.328,53.944,160.440
C04445=1007.946,315.753,-155.663,169.336,53.938,160.440
C04446=1007.951,316.000,-155.695,169.343,53.932,160.440
C04447=1007.957,316.249,-155.727,169.349,53.926,160.440
C04448=1007.962,316.497,-155.758,169.357,53.921,160.440
C04449=1007.968,316.744,-155.789,169.364,53.914,160.440
C04450=1007.974,316.992,-155.821,169.372,53.909,160.441
C04451=1007.978,317.240,-155.854,169.378,53.903,160.441
C04452=1007.984,317.489,-155.886,169.386,53.897,160.441
C04453=1007.990,317.736,-155.917,169.393,53.891,160.441
C04454=1007.995,317.984,-155.949,169.400,53.885,160.441
C04455=1008.001,318.232,-155.981,169.407,53.879,160.441
C04456=1008.006,318.480,-156.013,169.414,53.874,160.442
C04457=1008.012,318.728,-156.045,169.422,53.868,160.442
C04458=1008.017,318.975,-156.077,169.429,53.862,160.442
C04459=1008.022,319.223,-156.109,169.437,53.856,160.443
C04460=1008.028,319.471,-156.141,169.443,53.851,160.443
C04461=1008.034,319.719,-156.172,169.450,53.845,160.443
C04462=1008.039,319.967,-156.205,169.458,53.839,160.443
C04463=1008.045,320.215,-156.237,169.466,53.833,160.444
C04464=1008.051,320.462,-156.269,169.473,53.827,160.444
C04465=1008.057,320.710,-156.301,169.479,53.822,160.444
C04466=1008.062,320.958,-156.333,169.487,53.816,160.444
C04467=1008.068,321.206,-156.365,169.495,53.811,160.444
C04468=1008.073,321.454,-156.397,169.502,53.804,160.445
C04469=1008.079,321.702,-156.430,169.509,53.799,160.445
C04470=1008.085,321.950,-156.462,169.516,53.793,160.445
C04471=1008.090,322.197,-156.494,169.524,53.788,160.445
C04472=1008.096,322.445,-156.526,169.531,53.782,160.445
C04473=1008.102,322.693,-156.559,169.539,53.776,160.446
C04474=1008.107,322.941,-156.591,169.546,53.770,160.446
C04475=1008.113,323.189,-156.623,169.554,53.765,160.446
C04476=1008.120,323.437,-156.656,169.560,53.759,160.447
C04477=1008.128,323.780,-156.700,169.571,53.751,160.447
C04478=1008.135,324.125,-156.745,169.581,53.743,160.447
C04479=1008.143,324.469,-156.790,169.591,53.736,160.448
C04480=1008.152,324.812,-156.835,169.603,53.728,160.448
C04481=1008.157,325.060,-156.868,169.609,53.723,160.449
C04482=1008.163,325.309,-156.901,169.617,53.717,160.449
C04483=1008.169,325.556,-156.933,169.625,53.712,160.449
C04484=1008.174,325.803,-156.966,169.632,53.706,160.450
C04485=1008.180,326.051,-156.999,169.640,53.700,160.450
C04486=1008.186,326.299,-157.033,169.647,53.695,160.450
C04487=1008.191,326.547,-157.066,169.654,53.690,160.450
C04488=1008.197,326.795,-157.098,169.662,53.684,160.451
C04489=1008.202,327.042,-157.131,169.669,53.678,160.451
C04490=1008.208,327.290,-157.164,169.677,53.673,160.451
C04491=1008.214,327.538,-157.197,169.685,53.667,160.452
C04492=1008.220,327.786,-157.230,169.692,53.662,160.452
C04493=1008.225,328.034,-157.264,169.700,53.657,160.452
C04494=1008.231,328.281,-157.296,169.707,53.651,160.453
C04495=1008.237,328.529,-157.330,169.715,53.646,160.453
C04496=1008.243,328.777,-157.362,169.722,53.640,160.453
C04497=1008.249,329.025,-157.396,169.730,53.635,160.454
C04498=1008.254,329.272,-157.429,169.738,53.630,160.454
C04499=1008.261,329.520,-157.462,169.746,53.624,160.454
C04500=1008.267,329.767,-157.496,169.753,53.618,160.455
C04501=1008.272,330.015,-157.529,169.761,53.613,160.455
C04502=1008.278,330.263,-157.562,169.768,53.608,160.456
C04503=1008.284,330.511,-157.595,169.776,53.603,160.456
C04504=1008.290,330.758,-157.628,169.783,53.597,160.456
C04505=1008.296,331.006,-157.662,169.791,53.592,160.457
C04506=1008.302,331.253,-157.695,169.799,53.587,160.457
C04507=1008.307,331.501,-157.729,169.807,53.582,160.458
C04508=1008.313,331.749,-157.763,169.815,53.576,160.458
C04509=1008.319,331.996,-157.796,169.822,53.570,160.458
C04510=1008.325,332.244,-157.830,169.830,53.566,160.459
C04511=1008.331,332.492,-157.863,169.838,53.560,160.459
C04512=1008.337,332.739,-157.897,169.846,53.555,160.460
C04513=1008.343,332.987,-157.931,169.853,53.550,160.460
C04514=1008.349,333.235,-157.965,169.861,53.545,160.460
C04515=1008.354,333.483,-157.998,169.869,53.539,160.461
C04516=1008.360,333.730,-158.032,169.877,53.534,160.461
C04517=1008.366,333.978,-158.066,169.884,53.529,160.461
C04518=1008.372,334.226,-158.100,169.892,53.524,160.462
C04519=1008.379,334.473,-158.133,169.900,53.518,160.462
C04520=1008.384,334.721,-158.167,169.908,53.513,160.463
C04521=1008.391,334.969,-158.201,169.916,53.508,160.463
C04522=1008.397,335.216,-158.235,169.924,53.503,160.464
C04523=1008.402,335.463,-158.269,169.932,53.498,160.464
C04524=1008.409,335.712,-158.303,169.940,53.493,160.465
C04525=1008.414,335.959,-158.337,169.948,53.487,160.465
C04526=1008.420,336.206,-158.371,169.956,53.482,160.465
C04527=1008.427,336.454,-158.405,169.964,53.478,160.466
C04528=1008.433,336.701,-158.439,169.971,53.472,160.466
C04529=1008.439,336.949,-158.472,169.980,53.467,160.467
C04530=1008.445,337.197,-158.507,169.988,53.462,160.467
C04531=1008.451,337.444,-158.541,169.996,53.457,160.468
C04532=1008.458,337.692,-158.575,170.003,53.452,160.468
C04533=1008.464,337.940,-158.609,170.012,53.447,160.469
C04534=1008.469,338.187,-158.643,170.020,53.442,160.469
C04535=1008.476,338.434,-158.678,170.028,53.437,160.470
C04536=1008.481,338.682,-158.713,170.036,53.432,160.470
C04537=1008.490,339.022,-158.760,170.046,53.425,160.471
C04538=1008.498,339.361,-158.807,170.057,53.418,160.472
C04539=1008.507,339.701,-158.855,170.069,53.411,160.472
C04540=1008.516,340.041,-158.902,170.079,53.405,160.473
C04541=1008.521,340.288,-158.936,170.087,53.400,160.473
C04542=1008.528,340.535,-158.971,170.096,53.395,160.474
C04543=1008.533,340.783,-159.006,170.104,53.390,160.474
C04544=1008.540,341.031,-159.040,170.112,53.385,160.475
C04545=1008.547,341.278,-159.075,170.120,53.381,160.476
C04546=1008.552,341.526,-159.109,170.128,53.376,160.476
C04547=1008.559,341.773,-159.144,170.137,53.371,160.477
C04548=1008.565,342.021,-159.179,170.145,53.366,160.477
C04549=1008.571,342.268,-159.214,170.153,53.361,160.478
C04550=1008.578,342.516,-159.249,170.161,53.356,160.478
C04551=1008.584,342.763,-159.284,170.170,53.351,160.479
C04552=1008.589,343.011,-159.318,170.178,53.346,160.479
C04553=1008.596,343.258,-159.354,170.187,53.342,160.480
C04554=1008.603,343.506,-159.389,170.195,53.337,160.481
C04555=1008.609,343.754,-159.423,170.203,53.332,160.481
C04556=1008.616,344.000,-159.458,170.211,53.327,160.482
C04557=1008.622,344.248,-159.494,170.219,53.322,160.482
C04558=1008.628,344.496,-159.528,170.228,53.318,160.483
C04559=1008.635,344.743,-159.563,170.236,53.313,160.484
C04560=1008.642,344.991,-159.598,170.244,53.308,160.484
C04561=1008.647,345.238,-159.634,170.252,53.304,160.485
C04562=1008.654,345.485,-159.669,170.261,53.298,160.485
C04563=1008.661,345.732,-159.704,170.269,53.293,160.486
C04564=1008.667,345.980,-159.740,170.278,53.289,160.487
C04565=1008.673,346.227,-159.775,170.286,53.284,160.487
C04566=1008.680,346.475,-159.810,170.295,53.280,160.488
C04567=1008.686,346.722,-159.846,170.303,53.275,160.489
C04568=1008.693,346.970,-159.881,170.311,53.271,160.489
C04569=1008.699,347.218,-159.917,170.319,53.266,160.490
C04570=1008.706,347.465,-159.952,170.329,53.261,160.491
C04571=1008.711,347.712,-159.987,170.337,53.256,160.491
C04572=1008.718,347.959,-160.022,170.346,53.252,160.492
C04573=1008.724,348.207,-160.058,170.354,53.247,160.492
C04574=1008.732,348.454,-160.094,170.362,53.243,160.493
C04575=1008.738,348.702,-160.130,170.370,53.238,160.494
C04576=1008.745,348.949,-160.165,170.380,53.234,160.494
C04577=1008.751,349.197,-160.201,170.388,53.229,160.495
C04578=1008.758,349.444,-160.237,170.397,53.224,160.496
C04579=1008.764,349.691,-160.272,170.405,53.220,160.496
C04580=1008.771,349.938,-160.308,170.414,53.216,160.497
C04581=1008.777,350.186,-160.344,170.422,53.211,160.498
C04582=1008.784,350.433,-160.379,170.431,53.206,160.499
C04583=1008.790,350.680,-160.415,170.440,53.202,160.499
C04584=1008.797,350.928,-160.451,170.448,53.198,160.500
C04585=1008.804,351.175,-160.487,170.456,53.193,160.501
C04586=1008.810,351.423,-160.523,170.466,53.188,160.501
C04587=1008.817,351.670,-160.559,170.475,53.184,160.502
C04588=1008.823,351.917,-160.594,170.483,53.180,160.503
C04589=1008.831,352.165,-160.630,170.492,53.176,160.504
C04590=1008.837,352.412,-160.667,170.500,53.171,160.504
C04591=1008.843,352.659,-160.703,170.509,53.166,160.505
C04592=1008.851,352.906,-160.738,170.518,53.162,160.506
C04593=1008.857,353.154,-160.775,170.526,53.158,160.506
C04594=1008.864,353.401,-160.812,170.535,53.153,160.507
C04595=1008.870,353.648,-160.848,170.544,53.149,160.508
C04596=1008.878,353.896,-160.884,170.553,53.145,160.509
C04597=1008.885,354.194,-160.928,170.564,53.140,160.510
C04598=1008.894,354.493,-160.971,170.574,53.134,160.511
C04599=1008.902,354.792,-161.016,170.586,53.129,160.512
C04600=1008.910,355.090,-161.060,170.596,53.124,160.513
C04601=1008.918,355.338,-161.096,170.605,53.120,160.513
C04602=1008.924,355.585,-161.133,170.613,53.116,160.514
C04603=1008.931,355.832,-161.170,170.623,53.111,160.515
C04604=1008.938,356.079,-161.205,170.631,53.107,160.516
C04605=1008.945,356.327,-161.242,170.640,53.103,160.517
C04606=1008.951,356.574,-161.279,170.650,53.098,160.517
C04607=1008.958,356.822,-161.315,170.658,53.094,160.518
C04608=1008.965,357.068,-161.351,170.667,53.090,160.519
C04609=1008.642,354.940,-161.393,170.571,53.176,160.520
C04610=1008.636,354.694,-161.358,170.563,53.180,160.520
C04611=1008.628,354.447,-161.322,170.553,53.185,160.519
C04612=1008.622,354.202,-161.285,170.545,53.189,160.518
C04613=1008.615,353.955,-161.249,170.536,53.194,160.517
C04614=1008.608,353.708,-161.214,170.527,53.198,160.517
C04615=1008.601,353.461,-161.177,170.518,53.202,160.516
C04616=1008.595,353.213,-161.140,170.509,53.207,160.515
C04617=1008.589,352.966,-161.105,170.501,53.211,160.514
C04618=1008.581,352.718,-161.068,170.491,53.216,160.513
C04619=1008.575,352.471,-161.032,170.483,53.220,160.513
C04620=1008.569,352.224,-160.996,170.474,53.224,160.512
C04621=1008.562,351.977,-160.960,170.466,53.228,160.511
C04622=1008.556,351.730,-160.924,170.456,53.233,160.510
C04623=1008.548,351.482,-160.888,170.448,53.237,160.510
C04624=1008.541,351.235,-160.852,170.440,53.242,160.509
C04625=1008.535,350.987,-160.817,170.431,53.246,160.508
C04626=1008.528,350.740,-160.782,170.422,53.251,160.508
C04627=1008.522,350.493,-160.745,170.413,53.255,160.507
C04628=1008.515,350.246,-160.710,170.405,53.260,160.506
C04629=1008.508,349.998,-160.673,170.396,53.264,160.506
C04630=1008.501,349.750,-160.638,170.388,53.269,160.505
C04631=1008.495,349.503,-160.602,170.379,53.273,160.504
C04632=1008.488,349.256,-160.567,170.370,53.278,160.503
C04633=1008.482,349.008,-160.531,170.361,53.282,160.503
C04634=1008.476,348.761,-160.496,170.353,53.287,160.502
C04635=1008.470,348.513,-160.460,170.345,53.292,160.501
C04636=1008.463,348.266,-160.425,170.336,53.296,160.501
C04637=1008.456,348.019,-160.388,170.328,53.300,160.500
C04638=1008.450,347.772,-160.353,170.319,53.305,160.499
C04639=1008.444,347.524,-160.317,170.310,53.310,160.499
C04640=1008.437,347.276,-160.282,170.302,53.315,160.498
C04641=1008.431,347.029,-160.247,170.293,53.319,160.497
C04642=1008.425,346.782,-160.212,170.285,53.324,160.497
C04643=1008.419,346.534,-160.176,170.277,53.328,160.496
C04644=1008.412,346.287,-160.141,170.269,53.333,160.495
C04645=1008.405,346.040,-160.106,170.259,53.338,160.495
C04646=1008.399,345.792,-160.070,170.251,53.342,160.494
C04647=1008.392,345.545,-160.035,170.242,53.347,160.493
C04648=1008.386,345.297,-159.999,170.234,53.352,160.493
C04649=1008.380,345.050,-159.965,170.226,53.357,160.492
C04650=1008.374,344.802,-159.930,170.218,53.361,160.492
C04651=1008.367,344.555,-159.895,170.210,53.366,160.491
C04652=1008.361,344.307,-159.859,170.202,53.371,160.491
C04653=1008.354,344.059,-159.825,170.193,53.375,160.490
C04654=1008.348,343.813,-159.790,170.184,53.380,160.489
C04655=1008.341,343.565,-159.755,170.176,53.385,160.489
C04656=1008.335,343.317,-159.720,170.168,53.390,160.488
C04657=1008.330,343.070,-159.685,170.159,53.394,160.487
C04658=1008.323,342.822,-159.651,170.151,53.399,160.487
C04659=1008.316,342.575,-159.616,170.143,53.404,160.486
C04660=1008.310,342.327,-159.581,170.135,53.409,160.486
C04661=1008.304,342.080,-159.546,170.127,53.414,160.485
C04662=1008.298,341.832,-159.511,170.119,53.419,160.485
C04663=1008.292,341.585,-159.477,170.110,53.423,160.484
C04664=1008.285,341.337,-159.442,170.102,53.428,160.483
C04665=1008.279,341.089,-159.408,170.094,53.433,160.483
C04666=1008.273,340.842,-159.372,170.086,53.438,160.482
C04667=1008.267,340.594,-159.338,170.078,53.443,160.482
C04668=1008.261,340.347,-159.304,170.070,53.448,160.481
C04669=1008.254,340.100,-159.269,170.062,53.453,160.481
C04670=1008.246,339.758,-159.221,170.050,53.460,160.480
C04671=1008.237,339.416,-159.174,170.039,53.467,160.479
C04672=1008.229,339.074,-159.126,170.027,53.473,160.478
C04673=1008.221,338.732,-159.079,170.016,53.480,160.478
C04674=1008.214,338.484,-159.044,170.008,53.485,160.477
C04675=1008.209,338.237,-159.010,170.000,53.490,160.477
C04676=1008.203,337.990,-158.976,169.993,53.495,160.476
C04677=1008.197,337.741,-158.941,169.985,53.500,160.476
C04678=1008.191,337.494,-158.907,169.976,53.505,160.475
C04679=1008.185,337.246,-158.873,169.968,53.510,160.475
C04680=1008.179,336.999,-158.839,169.960,53.515,160.474
C04681=1008.172,336.752,-158.805,169.953,53.521,160.474
C04682=1008.166,336.504,-158.771,169.945,53.526,160.473
C04683=1008.160,336.257,-158.737,169.936,53.530,160.473
C04684=1008.154,336.009,-158.704,169.928,53.535,160.472
C04685=1008.148,335.761,-158.669,169.921,53.541,160.472
C04686=1008.142,335.513,-158.635,169.913,53.546,160.472
C04687=1008.136,335.266,-158.602,169.904,53.551,160.471
C04688=1008.131,335.018,-158.568,169.896,53.556,160.470
C04689=1008.124,334.770,-158.533,169.889,53.561,160.470
C04690=1008.118,334.523,-158.501,169.881,53.566,160.470
C04691=1008.112,334.275,-158.466,169.873,53.572,160.469
C04692=1008.106,334.028,-158.432,169.866,53.576,160.469
C04693=1008.100,333.780,-158.399,169.858,53.581,160.468
C04694=1008.094,333.532,-158.365,169.850,53.587,160.468
C04695=1008.089,333.284,-158.331,169.842,53.592,160.467
C04696=1008.083,333.037,-158.297,169.834,53.597,160.467
C04697=1008.077,332.789,-158.264,169.826,53.602,160.467
C04698=1008.071,332.542,-158.230,169.819,53.608,160.466
C04699=1008.065,332.294,-158.197,169.811,53.613,160.466
C04700=1008.059,332.047,-158.163,169.803,53.619,160.465
C04701=1008.053,331.798,-158.129,169.795,53.623,160.465
C04702=1008.047,331.550,-158.096,169.787,53.629,160.465
C04703=1008.042,331.303,-158.062,169.780,53.634,160.464
C04704=1008.036,331.055,-158.029,169.773,53.639,160.464
C04705=1008.030,330.808,-157.996,169.764,53.644,160.463
C04706=1008.024,330.560,-157.963,169.757,53.650,160.463
C04707=1008.018,330.313,-157.929,169.749,53.655,160.463
C04708=1008.012,330.065,-157.896,169.741,53.660,160.462
C04709=1008.006,329.817,-157.862,169.733,53.666,160.462
C04710=1008.001,329.569,-157.829,169.726,53.672,160.462
C04711=1007.995,329.322,-157.796,169.718,53.676,160.461
C04712=1007.989,329.074,-157.763,169.710,53.682,160.461
C04713=1007.983,328.826,-157.730,169.703,53.687,160.460
C04714=1007.977,328.578,-157.697,169.696,53.693,160.460
C04715=1007.972,328.331,-157.664,169.688,53.698,160.460
C04716=1007.966,328.083,-157.631,169.680,53.703,160.459
C04717=1007.960,327.835,-157.598,169.672,53.709,160.459
C04718=1007.955,327.588,-157.565,169.665,53.715,160.459
C04719=1007.949,327.340,-157.532,169.657,53.720,160.458
C04720=1007.943,327.092,-157.498,169.650,53.725,160.458
C04721=1007.938,326.843,-157.466,169.642,53.730,160.458
C04722=1007.932,326.597,-157.433,169.635,53.736,160.457
C04723=1007.927,326.349,-157.400,169.627,53.742,160.457
C04724=1007.920,326.101,-157.367,169.620,53.747,160.457
C04725=1007.915,325.853,-157.334,169.612,53.753,160.456
C04726=1007.909,325.605,-157.301,169.605,53.758,160.456
C04727=1007.904,325.358,-157.269,169.597,53.763,160.456
C04728=1007.898,325.110,-157.236,169.590,53.769,160.455
C04729=1007.893,324.862,-157.202,169.582,53.774,160.455
C04730=1007.884,324.515,-157.158,169.572,53.783,160.455
C04731=1007.876,324.169,-157.112,169.561,53.790,160.454
C04732=1007.868,323.823,-157.068,169.551,53.798,160.454
C04733=1007.860,323.477,-157.022,169.541,53.805,160.453
C04734=1007.855,323.229,-156.990,169.533,53.811,160.453
C04735=1007.849,322.981,-156.958,169.526,53.817,160.453
C04736=1007.843,322.734,-156.925,169.518,53.823,160.453
C04737=1007.837,322.486,-156.893,169.511,53.829,160.452
C04738=1007.831,322.237,-156.861,169.504,53.834,160.452
C04739=1007.826,321.990,-156.829,169.496,53.839,160.452
C04740=1007.820,321.742,-156.796,169.489,53.845,160.451
C04741=1007.815,321.494,-156.765,169.481,53.851,160.451
C04742=1007.809,321.246,-156.733,169.474,53.857,160.451
C04743=1007.803,320.999,-156.701,169.467,53.862,160.451
C04744=1007.797,320.751,-156.669,169.460,53.868,160.450
C04745=1007.792,320.503,-156.636,169.452,53.874,160.450
C04746=1007.786,320.255,-156.604,169.445,53.880,160.450
C04747=1007.780,320.007,-156.572,169.437,53.885,160.450
C04748=1007.775,319.759,-156.540,169.431,53.891,160.449
C04749=1007.770,319.512,-156.509,169.423,53.896,160.449
C04750=1007.764,319.264,-156.477,169.416,53.903,160.449
C04751=1007.759,319.016,-156.444,169.408,53.908,160.449
C04752=1007.753,318.768,-156.412,169.402,53.914,160.448
C04753=1007.748,318.520,-156.381,169.395,53.920,160.448
C04754=1007.742,318.272,-156.349,169.387,53.925,160.448
C04755=1007.736,318.024,-156.317,169.379,53.931,160.448
C04756=1007.732,317.777,-156.285,169.373,53.937,160.448
C04757=1007.726,317.528,-156.253,169.365,53.943,160.447
C04758=1007.721,317.280,-156.222,169.358,53.948,160.447
C04759=1007.715,317.033,-156.190,169.351,53.955,160.447
C04760=1007.709,316.784,-156.158,169.344,53.960,160.447
C04761=1007.704,316.537,-156.126,169.337,53.966,160.447
C04762=1007.699,316.289,-156.094,169.329,53.972,160.446
C04763=1007.693,316.041,-156.062,169.322,53.978,160.446
C04764=1007.688,315.793,-156.031,169.315,53.983,160.446
C04765=1007.683,315.545,-156.000,169.308,53.990,160.446
C04766=1007.677,315.298,-155.968,169.301,53.995,160.445
C04767=1007.672,315.049,-155.937,169.295,54.001,160.445
C04768=1007.667,314.801,-155.904,169.287,54.007,160.445
C04769=1007.662,314.554,-155.873,169.280,54.013,160.445
C04770=1007.656,314.306,-155.841,169.272,54.019,160.445
C04771=1007.651,314.058,-155.810,169.266,54.025,160.445
C04772=1007.646,313.810,-155.778,169.258,54.030,160.444
C04773=1007.640,313.562,-155.747,169.251,54.037,160.444
C04774=1007.635,313.314,-155.715,169.245,54.042,160.444
C04775=1007.630,313.066,-155.683,169.237,54.048,160.444
C04776=1007.625,312.818,-155.652,169.230,54.055,160.444
C04777=1007.620,312.571,-155.621,169.224,54.060,160.444
C04778=1007.614,312.323,-155.590,169.217,54.066,160.443
C04779=1007.609,312.075,-155.558,169.209,54.073,160.443
C04780=1007.605,311.827,-155.526,169.203,54.078,160.443
C04781=1007.599,311.579,-155.495,169.196,54.084,160.443
C04782=1007.594,311.331,-155.464,169.188,54.091,160.443
C04783=1007.589,311.083,-155.433,169.182,54.096,160.443
C04784=1007.584,310.835,-155.401,169.175,54.102,160.443
C04785=1007.579,310.587,-155.370,169.168,54.109,160.442
C04786=1007.574,310.339,-155.338,169.161,54.114,160.442
C04787=1007.569,310.091,-155.307,169.154,54.120,160.442
C04788=1007.564,309.843,-155.276,169.148,54.126,160.442
C04789=1007.559,309.596,-155.244,169.140,54.132,160.442
C04790=1007.552,309.255,-155.202,169.131,54.141,160.442
C04791=1007.545,308.915,-155.159,169.121,54.149,160.441
C04792=1007.538,308.573,-155.116,169.111,54.157,160.441
C04793=1007.531,308.233,-155.073,169.103,54.166,160.441
C04794=1007.527,307.986,-155.043,169.096,54.171,160.441
C04795=1007.521,307.738,-155.012,169.088,54.178,160.441
C04796=1007.515,307.490,-154.982,169.082,54.184,160.441
C04797=1007.510,307.242,-154.951,169.075,54.190,160.441
C04798=1007.505,306.993,-154.921,169.068,54.196,160.441
C04799=1007.500,306.746,-154.891,169.062,54.202,160.441
C04800=1007.494,306.498,-154.860,169.055,54.209,160.441
C04801=1007.489,306.250,-154.829,169.048,54.215,160.440
C04802=1007.484,306.001,-154.800,169.041,54.221,160.440
C04803=1007.479,305.753,-154.769,169.034,54.227,160.440
C04804=1007.474,305.505,-154.738,169.027,54.234,160.440
C04805=1007.469,305.257,-154.709,169.021,54.240,160.440
C04806=1007.464,305.009,-154.678,169.014,54.246,160.440
C04807=1007.458,304.762,-154.647,169.007,54.252,160.440
C04808=1007.453,304.513,-154.617,169.001,54.258,160.440
C04809=1007.448,304.266,-154.587,168.993,54.265,160.440
C04810=1007.443,304.017,-154.557,168.986,54.271,160.440
C04811=1007.437,303.769,-154.526,168.980,54.277,160.440
C04812=1007.432,303.521,-154.496,168.973,54.283,160.439
C04813=1007.427,303.273,-154.466,168.966,54.290,160.440
C04814=1007.420,302.912,-154.422,168.957,54.299,160.440
C04815=1007.412,302.550,-154.378,168.947,54.309,160.439
C04816=1007.404,302.189,-154.334,168.938,54.318,160.439
C04817=1007.397,301.828,-154.290,168.928,54.327,160.439
C04818=1007.155,302.488,-154.736,168.923,54.352,160.444
C04819=1007.159,302.715,-154.764,168.930,54.346,160.444
C04820=1007.163,302.940,-154.791,168.936,54.340,160.444
C04821=1007.169,303.166,-154.819,168.942,54.334,160.444
C04822=1007.173,303.391,-154.846,168.948,54.329,160.444
C04823=1007.177,303.618,-154.874,168.954,54.324,160.444
C04824=1007.182,303.844,-154.901,168.960,54.318,160.445
C04825=1007.187,304.069,-154.928,168.967,54.312,160.445
C04826=1007.191,304.296,-154.956,168.973,54.306,160.445
C04827=1007.197,304.544,-154.986,168.979,54.300,160.445
C04828=1007.201,304.793,-155.017,168.986,54.294,160.445
C04829=1007.207,305.040,-155.047,168.993,54.288,160.445
C04830=1007.211,305.288,-155.077,168.999,54.282,160.445
C04831=1007.217,305.536,-155.107,169.007,54.275,160.445
C04832=1007.222,305.784,-155.138,169.013,54.269,160.445
C04833=1007.227,306.032,-155.167,169.020,54.263,160.445
C04834=1007.232,306.280,-155.198,169.027,54.257,160.445
C04835=1007.238,306.528,-155.229,169.033,54.251,160.445
C04836=1007.243,306.777,-155.259,169.041,54.245,160.446
C04837=1007.249,307.025,-155.289,169.048,54.239,160.446
C04838=1007.254,307.273,-155.320,169.054,54.233,160.446
C04839=1007.259,307.520,-155.350,169.061,54.226,160.446
C04840=1007.264,307.768,-155.381,169.068,54.220,160.446
C04841=1007.270,308.016,-155.411,169.075,54.214,160.446
C04842=1007.275,308.265,-155.442,169.082,54.208,160.446
C04843=1007.281,308.607,-155.485,169.091,54.199,160.447
C04844=1007.288,308.949,-155.528,169.101,54.191,160.447
C04845=1007.295,309.292,-155.571,169.111,54.183,160.447
C04846=1007.302,309.635,-155.614,169.119,54.175,160.447
C04847=1007.307,309.883,-155.645,169.127,54.169,160.447
C04848=1007.312,310.131,-155.676,169.134,54.162,160.447
C04849=1007.317,310.380,-155.708,169.140,54.157,160.448
C04850=1007.322,310.627,-155.739,169.148,54.151,160.448
C04851=1007.327,310.875,-155.770,169.155,54.144,160.448
C04852=1007.332,311.123,-155.801,169.161,54.139,160.448
C04853=1007.338,311.371,-155.833,169.168,54.133,160.448
C04854=1007.342,311.619,-155.865,169.175,54.127,160.448
C04855=1007.347,311.867,-155.896,169.182,54.121,160.449
C04856=1007.352,312.115,-155.927,169.189,54.115,160.449
C04857=1007.358,312.362,-155.959,169.196,54.110,160.449
C04858=1007.363,312.611,-155.990,169.203,54.103,160.449
C04859=1007.368,312.859,-156.021,169.211,54.098,160.449
C04860=1007.373,313.107,-156.053,169.217,54.092,160.449
C04861=1007.378,313.354,-156.085,169.225,54.086,160.450
C04862=1007.383,313.602,-156.116,169.232,54.080,160.450
C04863=1007.388,313.850,-156.147,169.238,54.074,160.450
C04864=1007.393,314.098,-156.178,169.245,54.068,160.450
C04865=1007.399,314.345,-156.210,169.253,54.062,160.450
C04866=1007.403,314.594,-156.241,169.259,54.056,160.451
C04867=1007.409,314.842,-156.273,169.267,54.051,160.451
C04868=1007.415,315.090,-156.305,169.274,54.044,160.451
C04869=1007.420,315.338,-156.336,169.281,54.039,160.451
C04870=1007.425,315.585,-156.368,169.288,54.033,160.451
C04871=1007.430,315.833,-156.399,169.295,54.027,160.452
C04872=1007.435,316.082,-156.431,169.303,54.021,160.452
C04873=1007.441,316.329,-156.463,169.309,54.016,160.452
C04874=1007.446,316.577,-156.495,169.317,54.010,160.452
C04875=1007.452,316.824,-156.526,169.324,54.004,160.452
C04876=1007.458,317.073,-156.558,169.331,53.998,160.453
C04877=1007.463,317.321,-156.589,169.338,53.993,160.453
C04878=1007.467,317.569,-156.621,169.345,53.986,160.453
C04879=1007.473,317.817,-156.653,169.353,53.981,160.454
C04880=1007.479,318.064,-156.685,169.360,53.975,160.454
C04881=1007.484,318.312,-156.717,169.367,53.969,160.454
C04882=1007.490,318.560,-156.749,169.374,53.964,160.454
C04883=1007.495,318.807,-156.780,169.382,53.958,160.455
C04884=1007.500,319.055,-156.813,169.388,53.952,160.454
C04885=1007.506,319.304,-156.845,169.396,53.946,160.455
C04886=1007.511,319.551,-156.876,169.403,53.941,160.455
C04887=1007.517,319.799,-156.908,169.411,53.935,160.456
C04888=1007.523,320.047,-156.940,169.418,53.930,160.456
C04889=1007.528,320.295,-156.973,169.425,53.923,160.456
C04890=1007.533,320.543,-157.004,169.432,53.918,160.456
C04891=1007.539,320.791,-157.036,169.440,53.912,160.457
C04892=1007.545,321.039,-157.068,169.447,53.907,160.457
C04893=1007.551,321.287,-157.100,169.454,53.901,160.457
C04894=1007.556,321.534,-157.132,169.462,53.896,160.457
C04895=1007.561,321.783,-157.164,169.469,53.889,160.457
C04896=1007.567,322.030,-157.196,169.477,53.884,160.458
C04897=1007.573,322.278,-157.229,169.483,53.878,160.458
C04898=1007.579,322.526,-157.261,169.491,53.873,160.458
C04899=1007.584,322.774,-157.292,169.499,53.867,160.459
C04900=1007.590,323.022,-157.324,169.506,53.862,160.459
C04901=1007.595,323.269,-157.357,169.514,53.856,160.459
C04902=1007.601,323.517,-157.389,169.521,53.851,160.460
C04903=1007.610,323.866,-157.435,169.532,53.843,160.460
C04904=1007.617,324.215,-157.480,169.542,53.835,160.461
C04905=1007.626,324.563,-157.526,169.553,53.827,160.461
C04906=1007.634,324.912,-157.571,169.563,53.819,160.461
C04907=1007.639,325.159,-157.604,169.570,53.814,160.462
C04908=1007.645,325.408,-157.637,169.578,53.808,160.462
C04909=1007.651,325.655,-157.669,169.585,53.803,160.462
C04910=1007.656,325.902,-157.702,169.593,53.798,160.463
C04911=1007.661,326.150,-157.736,169.600,53.792,160.463
C04912=1007.667,326.398,-157.768,169.608,53.787,160.463
C04913=1007.673,326.646,-157.801,169.616,53.781,160.464
C04914=1007.679,326.893,-157.834,169.623,53.775,160.464
C04915=1007.684,327.141,-157.867,169.630,53.771,160.465
C04916=1007.690,327.389,-157.900,169.638,53.765,160.465
C04917=1007.696,327.637,-157.932,169.646,53.759,160.465
C04918=1007.701,327.885,-157.966,169.653,53.754,160.465
C04919=1007.707,328.133,-157.999,169.661,53.749,160.466
C04920=1007.713,328.380,-158.031,169.669,53.743,160.466
C04921=1007.718,328.628,-158.065,169.676,53.738,160.467
C04922=1007.724,328.876,-158.097,169.684,53.733,160.467
C04923=1007.730,329.123,-158.131,169.691,53.727,160.467
C04924=1007.735,329.371,-158.164,169.699,53.722,160.468
C04925=1007.742,329.619,-158.197,169.707,53.717,160.468
C04926=1007.747,329.867,-158.230,169.715,53.711,160.469
C04927=1007.753,330.115,-158.263,169.722,53.706,160.469
C04928=1007.759,330.362,-158.296,169.730,53.701,160.470
C04929=1007.765,330.610,-158.330,169.737,53.696,160.470
C04930=1007.770,330.858,-158.363,169.745,53.691,160.470
C04931=1007.777,331.105,-158.396,169.753,53.685,160.471
C04932=1007.782,331.353,-158.430,169.760,53.679,160.471
C04933=1007.788,331.601,-158.463,169.769,53.674,160.471
C04934=1007.794,331.848,-158.497,169.776,53.669,160.472
C04935=1007.799,332.096,-158.530,169.784,53.664,160.472
C04936=1007.805,332.344,-158.564,169.792,53.659,160.473
C04937=1007.811,332.591,-158.598,169.800,53.653,160.473
C04938=1007.817,332.839,-158.631,169.807,53.649,160.474
C04939=1007.823,333.086,-158.665,169.815,53.643,160.474
C04940=1007.829,333.334,-158.698,169.823,53.638,160.474
C04941=1007.835,333.582,-158.732,169.830,53.633,160.475
C04942=1007.841,333.830,-158.766,169.839,53.628,160.475
C04943=1007.846,334.077,-158.800,169.847,53.623,160.476
C04944=1007.852,334.325,-158.833,169.854,53.617,160.476
C04945=1007.858,334.572,-158.867,169.862,53.612,160.477
C04946=1007.863,334.820,-158.900,169.871,53.607,160.477
C04947=1007.871,335.068,-158.934,169.878,53.602,160.478
C04948=1007.876,335.315,-158.968,169.886,53.597,160.478
C04949=1007.882,335.563,-159.002,169.894,53.592,160.479
C04950=1007.888,335.810,-159.036,169.902,53.587,160.479
C04951=1007.894,336.058,-159.070,169.910,53.581,160.480
C04952=1007.900,336.306,-159.103,169.918,53.576,160.480
C04953=1007.906,336.554,-159.138,169.926,53.571,160.481
C04954=1007.912,336.802,-159.172,169.933,53.567,160.481
C04955=1007.918,337.049,-159.206,169.941,53.562,160.482
C04956=1007.924,337.296,-159.239,169.949,53.556,160.482
C04957=1007.931,337.544,-159.273,169.957,53.551,160.482
C04958=1007.936,337.792,-159.308,169.965,53.546,160.483
C04959=1007.942,338.039,-159.342,169.973,53.542,160.484
C04960=1007.948,338.287,-159.376,169.981,53.537,160.484
C04961=1007.954,338.535,-159.410,169.990,53.532,160.485
C04962=1007.961,338.782,-159.445,169.998,53.527,160.485
C04963=1007.968,339.072,-159.485,170.008,53.521,160.486
C04964=1007.974,339.363,-159.526,170.016,53.515,160.486
C04965=1007.982,339.653,-159.566,170.027,53.509,160.487
C04966=1007.989,339.943,-159.606,170.037,53.504,160.488
C04967=1007.995,340.190,-159.641,170.045,53.499,160.488
C04968=1008.001,340.438,-159.676,170.053,53.494,160.489
C04969=1008.007,340.685,-159.710,170.061,53.489,160.489
C04970=1008.013,340.933,-159.744,170.069,53.484,160.490
C04971=1008.020,341.180,-159.779,170.077,53.479,160.490
C04972=1008.026,341.428,-159.813,170.085,53.474,160.491
C04973=1008.031,341.675,-159.848,170.093,53.469,160.492
C04974=1008.038,341.923,-159.883,170.101,53.464,160.492
C04975=1008.044,342.171,-159.917,170.110,53.460,160.493
C04976=1008.051,342.417,-159.952,170.118,53.455,160.493
C04977=1008.057,342.665,-159.987,170.126,53.450,160.494
C04978=1008.063,342.913,-160.022,170.134,53.445,160.494
C04979=1008.069,343.160,-160.056,170.143,53.441,160.495
C04980=1008.076,343.408,-160.092,170.151,53.436,160.496
C04981=1008.082,343.656,-160.126,170.159,53.431,160.496
C04982=1008.088,343.903,-160.161,170.167,53.426,160.497
C04983=1008.094,344.151,-160.196,170.176,53.422,160.498
C04984=1008.101,344.398,-160.231,170.185,53.417,160.498
C04985=1008.108,344.645,-160.266,170.193,53.412,160.499
C04986=1008.113,344.893,-160.300,170.201,53.407,160.499
C04987=1008.119,345.140,-160.336,170.209,53.402,160.500
C04988=1008.126,345.388,-160.371,170.218,53.398,160.501
C04989=1008.133,345.635,-160.406,170.226,53.393,160.501
C04990=1008.139,345.883,-160.442,170.234,53.388,160.502
C04991=1008.145,346.129,-160.477,170.243,53.384,160.503
C04992=1008.151,346.378,-160.512,170.251,53.379,160.503
C04993=1008.158,346.625,-160.547,170.260,53.374,160.504
C04994=1008.164,346.873,-160.582,170.269,53.370,160.504
C04995=1008.170,347.120,-160.618,170.277,53.365,160.505
C04996=1008.177,347.367,-160.653,170.286,53.361,160.506
C04997=1008.183,347.615,-160.688,170.294,53.356,160.507
C04998=1008.190,347.862,-160.724,170.302,53.352,160.507
C04999=1008.196,348.109,-160.760,170.310,53.347,160.508
C05000=1008.203,348.356,-160.795,170.320,53.342,160.509
C05001=1008.209,348.604,-160.831,170.329,53.338,160.509
C05002=1008.215,348.851,-160.866,170.337,53.333,160.510
C05003=1008.221,349.099,-160.901,170.345,53.329,160.511
C05004=1008.228,349.346,-160.937,170.354,53.325,160.511
C05005=1008.234,349.593,-160.973,170.362,53.320,160.512
C05006=1008.242,349.841,-161.008,170.371,53.315,160.513
C05007=1008.248,350.089,-161.044,170.380,53.311,160.514
C05008=1008.255,350.336,-161.080,170.388,53.307,160.514
C05009=1008.261,350.583,-161.116,170.397,53.302,160.515
C05010=1008.268,350.830,-161.152,170.405,53.297,160.516
C05011=1008.274,351.078,-161.187,170.415,53.293,160.516
C05012=1008.281,351.325,-161.223,170.423,53.288,160.517
C05013=1008.287,351.572,-161.259,170.432,53.284,160.518
C05014=1008.295,351.820,-161.294,170.440,53.280,160.519
C05015=1008.301,352.067,-161.331,170.450,53.275,160.520
C05016=1008.308,352.315,-161.366,170.458,53.271,160.520
C05017=1008.314,352.562,-161.402,170.467,53.267,160.521
C05018=1008.320,352.809,-161.439,170.476,53.263,160.522
C05019=1008.000,350.672,-161.486,170.381,53.347,160.523
C05020=1007.994,350.425,-161.450,170.372,53.351,160.522
C05021=1007.988,350.177,-161.415,170.364,53.356,160.521
C05022=1007.981,349.930,-161.379,170.355,53.361,160.521
C05023=1007.975,349.683,-161.344,170.346,53.365,160.520
C05024=1007.968,349.435,-161.308,170.337,53.369,160.519
C05025=1007.962,349.188,-161.273,170.329,53.374,160.518
C05026=1007.955,348.941,-161.236,170.321,53.379,160.518
C05027=1007.949,348.693,-161.201,170.312,53.383,160.517
C05028=1007.943,348.446,-161.166,170.303,53.388,160.516
C05029=1007.936,348.198,-161.130,170.294,53.392,160.515
C05030=1007.930,347.951,-161.095,170.286,53.397,160.515
C05031=1007.923,347.703,-161.060,170.278,53.401,160.514
C05032=1007.917,347.456,-161.024,170.269,53.406,160.514
C05033=1007.910,347.208,-160.989,170.261,53.410,160.513
C05034=1007.903,346.961,-160.954,170.251,53.415,160.512
C05035=1007.897,346.713,-160.918,170.243,53.420,160.511
C05036=1007.891,346.467,-160.883,170.235,53.424,160.511
C05037=1007.885,346.219,-160.847,170.227,53.429,160.510
C05038=1007.878,345.972,-160.812,170.218,53.433,160.509
C05039=1007.872,345.724,-160.776,170.210,53.438,160.509
C05040=1007.866,345.476,-160.742,170.201,53.442,160.508
C05041=1007.860,345.229,-160.707,170.193,53.447,160.508
C05042=1007.854,344.982,-160.672,170.185,53.452,160.507
C05043=1007.847,344.734,-160.637,170.176,53.457,160.506
C05044=1007.841,344.486,-160.602,170.167,53.461,160.505
C05045=1007.834,344.240,-160.567,170.159,53.466,160.505
C05046=1007.829,343.991,-160.532,170.151,53.471,160.504
C05047=1007.822,343.744,-160.497,170.142,53.475,160.503
C05048=1007.816,343.497,-160.463,170.134,53.480,160.503
C05049=1007.809,343.249,-160.428,170.126,53.485,160.502
C05050=1007.803,343.001,-160.393,170.118,53.489,160.502
C05051=1007.797,342.754,-160.358,170.109,53.494,160.501
C05052=1007.791,342.506,-160.324,170.101,53.499,160.501
C05053=1007.785,342.260,-160.289,170.093,53.504,160.500
C05054=1007.778,342.012,-160.255,170.085,53.508,160.499
C05055=1007.773,341.763,-160.220,170.077,53.513,160.499
C05056=1007.766,341.517,-160.185,170.069,53.518,160.498
C05057=1007.760,341.269,-160.150,170.060,53.523,160.498
C05058=1007.754,341.021,-160.116,170.052,53.528,160.497
C05059=1007.747,340.774,-160.081,170.043,53.534,160.497
C05060=1007.742,340.531,-160.048,170.036,53.537,160.496
C05061=1007.736,340.289,-160.014,170.028,53.542,160.495
C05062=1007.730,340.046,-159.980,170.019,53.547,160.495
C05063=1007.724,339.802,-159.946,170.011,53.552,160.494
C05064=1007.718,339.560,-159.913,170.003,53.557,160.494
C05065=1007.712,339.318,-159.879,169.995,53.562,160.493
C05066=1007.706,339.074,-159.845,169.988,53.567,160.493
C05067=1007.701,338.832,-159.811,169.980,53.572,160.492
C05068=1007.694,338.584,-159.777,169.972,53.576,160.492
C05069=1007.688,338.337,-159.743,169.964,53.581,160.491
C05070=1007.682,338.089,-159.708,169.956,53.586,160.491
C05071=1007.676,337.842,-159.674,169.948,53.591,160.490
C05072=1007.671,337.594,-159.640,169.940,53.596,160.489
C05073=1007.664,337.346,-159.605,169.931,53.601,160.489
C05074=1007.658,337.099,-159.573,169.923,53.606,160.488
C05075=1007.652,336.851,-159.539,169.915,53.611,160.488
C05076=1007.646,336.604,-159.504,169.907,53.616,160.487
C05077=1007.640,336.356,-159.470,169.899,53.621,160.487
C05078=1007.634,336.108,-159.437,169.891,53.627,160.486
C05079=1007.628,335.861,-159.403,169.883,53.631,160.486
C05080=1007.623,335.614,-159.369,169.875,53.636,160.485
C05081=1007.616,335.365,-159.335,169.867,53.641,160.485
C05082=1007.611,335.118,-159.301,169.859,53.646,160.484
C05083=1007.604,334.870,-159.268,169.851,53.652,160.484
C05084=1007.598,334.623,-159.234,169.844,53.656,160.483
C05085=1007.593,334.375,-159.201,169.836,53.661,160.483
C05086=1007.586,334.127,-159.166,169.828,53.666,160.482
C05087=1007.581,333.879,-159.133,169.820,53.672,160.482
C05088=1007.575,333.632,-159.099,169.812,53.677,160.481
C05089=1007.569,333.384,-159.066,169.804,53.682,160.481
C05090=1007.564,333.137,-159.032,169.797,53.687,160.481
C05091=1007.558,332.889,-158.998,169.788,53.692,160.480
C05092=1007.551,332.642,-158.965,169.781,53.698,160.480
C05093=1007.546,332.394,-158.931,169.773,53.703,160.479
C05094=1007.540,332.146,-158.898,169.765,53.708,160.479
C05095=1007.534,331.899,-158.864,169.758,53.713,160.478
C05096=1007.529,331.651,-158.831,169.750,53.718,160.478
C05097=1007.523,331.403,-158.797,169.742,53.724,160.478
C05098=1007.518,331.155,-158.764,169.734,53.729,160.477
C05099=1007.512,330.908,-158.730,169.727,53.734,160.477
C05100=1007.506,330.660,-158.697,169.718,53.739,160.476
C05101=1007.500,330.412,-158.664,169.711,53.745,160.476
C05102=1007.494,330.165,-158.631,169.703,53.750,160.475
C05103=1007.488,329.917,-158.598,169.696,53.755,160.475
C05104=1007.483,329.669,-158.564,169.688,53.760,160.474
C05105=1007.476,329.421,-158.532,169.680,53.766,160.474
C05106=1007.471,329.173,-158.498,169.673,53.771,160.474
C05107=1007.465,328.925,-158.465,169.665,53.776,160.473
C05108=1007.459,328.678,-158.432,169.657,53.782,160.473
C05109=1007.454,328.431,-158.399,169.649,53.787,160.473
C05110=1007.449,328.182,-158.367,169.642,53.792,160.472
C05111=1007.442,327.934,-158.334,169.635,53.798,160.472
C05112=1007.437,327.686,-158.301,169.627,53.803,160.472
C05113=1007.431,327.439,-158.268,169.619,53.808,160.471
C05114=1007.425,327.191,-158.235,169.611,53.814,160.471
C05115=1007.420,326.944,-158.202,169.605,53.819,160.470
C05116=1007.414,326.696,-158.170,169.597,53.824,160.470
C05117=1007.409,326.448,-158.136,169.589,53.830,160.470
C05118=1007.403,326.200,-158.103,169.581,53.835,160.469
C05119=1007.398,325.952,-158.071,169.574,53.841,160.469
C05120=1007.392,325.704,-158.038,169.566,53.847,160.469
C05121=1007.386,325.456,-158.004,169.559,53.851,160.468
C05122=1007.381,325.209,-157.973,169.551,53.857,160.468
C05123=1007.376,324.961,-157.939,169.544,53.862,160.467
C05124=1007.368,324.610,-157.894,169.534,53.870,160.467
C05125=1007.359,324.259,-157.848,169.522,53.878,160.466
C05126=1007.351,323.908,-157.802,169.512,53.885,160.466
C05127=1007.343,323.558,-157.757,169.501,53.894,160.466
C05128=1007.337,323.310,-157.725,169.494,53.900,160.465
C05129=1007.331,323.062,-157.692,169.487,53.905,160.465
C05130=1007.326,322.814,-157.660,169.480,53.910,160.465
C05131=1007.321,322.566,-157.628,169.472,53.916,160.464
C05132=1007.315,322.318,-157.596,169.464,53.922,160.464
C05133=1007.309,322.070,-157.564,169.457,53.927,160.464
C05134=1007.303,321.822,-157.532,169.450,53.933,160.464
C05135=1007.297,321.575,-157.500,169.442,53.938,160.463
C05136=1007.292,321.327,-157.467,169.435,53.944,160.463
C05137=1007.287,321.079,-157.435,169.427,53.950,160.462
C05138=1007.281,320.831,-157.403,169.421,53.955,160.462
C05139=1007.275,320.583,-157.372,169.413,53.960,160.462
C05140=1007.270,320.336,-157.340,169.405,53.966,160.462
C05141=1007.264,320.088,-157.308,169.398,53.972,160.461
C05142=1007.259,319.840,-157.276,169.391,53.977,160.461
C05143=1007.253,319.592,-157.244,169.384,53.983,160.461
C05144=1007.248,319.344,-157.212,169.376,53.989,160.461
C05145=1007.243,319.097,-157.180,169.369,53.995,160.460
C05146=1007.237,318.848,-157.148,169.362,54.000,160.460
C05147=1007.232,318.600,-157.117,169.354,54.005,160.460
C05148=1007.226,318.352,-157.085,169.347,54.012,160.460
C05149=1007.221,318.104,-157.053,169.341,54.017,160.459
C05150=1007.216,317.857,-157.022,169.333,54.023,160.459
C05151=1007.210,317.609,-156.990,169.325,54.028,160.459
C05152=1007.204,317.361,-156.958,169.318,54.035,160.458
C05153=1007.200,317.112,-156.926,169.312,54.040,160.458
C05154=1007.195,316.865,-156.895,169.304,54.046,160.458
C05155=1007.189,316.617,-156.863,169.296,54.051,160.458
C05156=1007.183,316.369,-156.831,169.290,54.057,160.458
C05157=1007.178,316.121,-156.800,169.283,54.063,160.457
C05158=1007.173,315.874,-156.768,169.275,54.069,160.457
C05159=1007.168,315.626,-156.736,169.269,54.074,160.457
C05160=1007.162,315.377,-156.705,169.261,54.080,160.457
C05161=1007.157,315.129,-156.673,169.254,54.086,160.456
C05162=1007.152,314.882,-156.641,169.247,54.092,160.456
C05163=1007.146,314.634,-156.610,169.240,54.097,160.456
C05164=1007.141,314.386,-156.579,169.233,54.104,160.456
C05165=1007.137,314.138,-156.547,169.226,54.109,160.455
C05166=1007.131,313.890,-156.516,169.219,54.115,160.455
C05167=1007.126,313.642,-156.485,169.211,54.121,160.455
C05168=1007.121,313.395,-156.453,169.205,54.127,160.455
C05169=1007.116,313.147,-156.422,169.197,54.133,160.455
C05170=1007.110,312.899,-156.390,169.190,54.138,160.454
C05171=1007.106,312.651,-156.359,169.184,54.144,160.454
C05172=1007.100,312.402,-156.327,169.176,54.150,160.454
C05173=1007.095,312.154,-156.296,169.169,54.156,160.454
C05174=1007.091,311.907,-156.265,169.163,54.162,160.454
C05175=1007.085,311.659,-156.234,169.155,54.168,160.453
C05176=1007.081,311.411,-156.202,169.149,54.174,160.453
C05177=1007.076,311.163,-156.171,169.141,54.179,160.453
C05178=1007.070,310.915,-156.140,169.134,54.186,160.453
C05179=1007.065,310.667,-156.109,169.128,54.191,160.453
C05180=1007.060,310.419,-156.078,169.120,54.197,160.453
C05181=1007.055,310.171,-156.046,169.114,54.203,160.453
C05182=1007.050,309.923,-156.014,169.107,54.209,160.452
C05183=1007.045,309.675,-155.983,169.099,54.215,160.452
C05184=1007.038,309.331,-155.940,169.090,54.224,160.452
C05185=1007.032,308.985,-155.897,169.080,54.232,160.452
C05186=1007.025,308.640,-155.853,169.071,54.240,160.451
C05187=1007.018,308.295,-155.811,169.062,54.248,160.451
C05188=1007.014,308.046,-155.779,169.055,54.254,160.451
C05189=1007.008,307.799,-155.749,169.047,54.261,160.451
C05190=1007.002,307.551,-155.719,169.041,54.266,160.451
C05191=1006.997,307.303,-155.688,169.034,54.272,160.451
C05192=1006.992,307.055,-155.658,169.028,54.278,160.451
C05193=1006.987,306.807,-155.628,169.020,54.285,160.450
C05194=1006.982,306.560,-155.598,169.013,54.291,160.450
C05195=1006.977,306.311,-155.567,169.007,54.297,160.450
C05196=1006.971,306.063,-155.537,168.999,54.303,160.450
C05197=1006.966,305.814,-155.507,168.993,54.309,160.450
C05198=1006.961,305.567,-155.477,168.986,54.315,160.450
C05199=1006.956,305.319,-155.446,168.979,54.322,160.450
C05200=1006.950,305.071,-155.416,168.973,54.327,160.450
C05201=1006.945,304.822,-155.385,168.966,54.334,160.450
C05202=1006.941,304.574,-155.355,168.960,54.340,160.450
C05203=1006.935,304.327,-155.325,168.953,54.346,160.449
C05204=1006.930,304.027,-155.288,168.944,54.353,160.449
C05205=1006.923,303.728,-155.253,168.936,54.361,160.449
C05206=1006.918,303.429,-155.216,168.928,54.368,160.449
C05207=1006.911,303.131,-155.180,168.920,54.376,160.449
C05208=1006.667,303.750,-155.621,168.916,54.398,160.453
C05209=1006.676,304.150,-155.670,168.926,54.389,160.453
C05210=1006.684,304.549,-155.718,168.937,54.379,160.453
C05211=1006.692,304.949,-155.766,168.948,54.369,160.454
C05212=1006.701,305.349,-155.815,168.960,54.359,160.454
C05213=1006.705,305.597,-155.845,168.966,54.353,160.454
C05214=1006.711,305.845,-155.876,168.973,54.347,160.454
C05215=1006.715,306.094,-155.906,168.979,54.341,160.454
C05216=1006.721,306.342,-155.936,168.987,54.335,160.455
C05217=1006.725,306.590,-155.966,168.994,54.329,160.455
C05218=1006.731,306.837,-155.996,169.000,54.323,160.455
C05219=1006.736,307.086,-156.027,169.007,54.317,160.455
C05220=1006.741,307.334,-156.058,169.014,54.311,160.455
C05221=1006.746,307.581,-156.088,169.021,54.305,160.455
C05222=1006.752,307.829,-156.118,169.028,54.298,160.455
C05223=1006.757,308.077,-156.149,169.035,54.293,160.456
C05224=1006.762,308.325,-156.179,169.042,54.287,160.456
C05225=1006.769,308.673,-156.223,169.051,54.279,160.456
C05226=1006.776,309.020,-156.266,169.061,54.270,160.456
C05227=1006.782,309.368,-156.310,169.071,54.262,160.457
C05228=1006.790,309.715,-156.354,169.081,54.254,160.457
C05229=1006.795,309.963,-156.385,169.087,54.248,160.457
C05230=1006.798,310.211,-156.416,169.094,54.242,160.457
C05231=1006.803,310.459,-156.447,169.100,54.236,160.457
C05232=1006.809,310.707,-156.478,169.108,54.231,160.458
C05233=1006.814,310.955,-156.509,169.114,54.225,160.457
C05234=1006.819,311.203,-156.540,169.122,54.219,160.458
C05235=1006.823,311.451,-156.572,169.129,54.213,160.458
C05236=1006.828,311.699,-156.603,169.136,54.207,160.458
C05237=1006.834,311.947,-156.634,169.143,54.201,160.458
C05238=1006.839,312.195,-156.665,169.149,54.196,160.459
C05239=1006.844,312.442,-156.697,169.157,54.189,160.459
C05240=1006.849,312.691,-156.728,169.164,54.184,160.459
C05241=1006.854,312.939,-156.760,169.170,54.178,160.459
C05242=1006.859,313.186,-156.791,169.178,54.172,160.459
C05243=1006.864,313.435,-156.822,169.186,54.166,160.460
C05244=1006.870,313.682,-156.854,169.192,54.160,160.460
C05245=1006.875,313.930,-156.885,169.199,54.155,160.460
C05246=1006.880,314.178,-156.916,169.205,54.149,160.460
C05247=1006.884,314.426,-156.948,169.213,54.143,160.461
C05248=1006.890,314.674,-156.980,169.221,54.137,160.461
C05249=1006.895,314.922,-157.011,169.227,54.131,160.461
C05250=1006.900,315.169,-157.042,169.235,54.126,160.461
C05251=1006.905,315.417,-157.073,169.242,54.120,160.462
C05252=1006.911,315.665,-157.105,169.248,54.114,160.462
C05253=1006.916,315.914,-157.137,169.256,54.108,160.462
C05254=1006.921,316.162,-157.168,169.264,54.103,160.462
C05255=1006.926,316.409,-157.200,169.270,54.098,160.463
C05256=1006.931,316.657,-157.231,169.277,54.091,160.463
C05257=1006.937,316.905,-157.263,169.285,54.086,160.463
C05258=1006.942,317.153,-157.295,169.292,54.080,160.463
C05259=1006.948,317.401,-157.327,169.299,54.075,160.464
C05260=1006.953,317.649,-157.358,169.306,54.068,160.464
C05261=1006.958,317.896,-157.390,169.313,54.063,160.464
C05262=1006.964,318.145,-157.422,169.321,54.057,160.464
C05263=1006.969,318.392,-157.453,169.328,54.052,160.465
C05264=1006.974,318.640,-157.486,169.335,54.046,160.465
C05265=1006.979,318.888,-157.516,169.342,54.041,160.465
C05266=1006.985,319.136,-157.549,169.350,54.034,160.465
C05267=1006.990,319.384,-157.580,169.357,54.029,160.466
C05268=1006.996,319.632,-157.612,169.364,54.024,160.466
C05269=1007.002,319.880,-157.644,169.372,54.018,160.466
C05270=1007.006,320.127,-157.676,169.379,54.012,160.467
C05271=1007.012,320.376,-157.708,169.386,54.007,160.467
C05272=1007.018,320.623,-157.740,169.393,54.001,160.467
C05273=1007.024,320.871,-157.772,169.401,53.996,160.468
C05274=1007.029,321.119,-157.803,169.409,53.990,160.468
C05275=1007.034,321.367,-157.836,169.415,53.985,160.468
C05276=1007.040,321.615,-157.868,169.423,53.979,160.469
C05277=1007.045,321.862,-157.899,169.431,53.973,160.469
C05278=1007.051,322.111,-157.931,169.438,53.968,160.469
C05279=1007.057,322.358,-157.963,169.445,53.963,160.469
C05280=1007.063,322.606,-157.995,169.452,53.957,160.470
C05281=1007.068,322.855,-158.028,169.460,53.951,160.470
C05282=1007.074,323.102,-158.060,169.468,53.946,160.470
C05283=1007.080,323.350,-158.092,169.475,53.940,160.471
C05284=1007.085,323.598,-158.124,169.482,53.935,160.471
C05285=1007.093,323.951,-158.170,169.493,53.927,160.472
C05286=1007.101,324.304,-158.215,169.503,53.919,160.472
C05287=1007.110,324.658,-158.261,169.514,53.911,160.473
C05288=1007.117,325.011,-158.308,169.525,53.904,160.473
C05289=1007.122,325.258,-158.341,169.532,53.898,160.473
C05290=1007.128,325.506,-158.373,169.540,53.893,160.474
C05291=1007.134,325.754,-158.407,169.548,53.888,160.474
C05292=1007.139,326.001,-158.439,169.556,53.882,160.475
C05293=1007.145,326.250,-158.472,169.562,53.877,160.475
C05294=1007.150,326.498,-158.505,169.570,53.871,160.475
C05295=1007.156,326.744,-158.537,169.578,53.866,160.476
C05296=1007.161,326.993,-158.570,169.586,53.860,160.476
C05297=1007.167,327.241,-158.603,169.592,53.855,160.476
C05298=1007.173,327.488,-158.636,169.600,53.850,160.477
C05299=1007.178,327.736,-158.669,169.608,53.845,160.477
C05300=1007.183,327.984,-158.702,169.616,53.839,160.478
C05301=1007.190,328.232,-158.734,169.624,53.834,160.478
C05302=1007.195,328.480,-158.768,169.631,53.828,160.478
C05303=1007.201,328.727,-158.800,169.638,53.824,160.479
C05304=1007.207,328.975,-158.834,169.646,53.818,160.479
C05305=1007.212,329.222,-158.867,169.654,53.813,160.480
C05306=1007.218,329.470,-158.899,169.662,53.808,160.480
C05307=1007.224,329.718,-158.933,169.669,53.802,160.480
C05308=1007.229,329.966,-158.965,169.678,53.797,160.481
C05309=1007.235,330.214,-158.998,169.684,53.792,160.481
C05310=1007.241,330.462,-159.031,169.692,53.787,160.482
C05311=1007.246,330.710,-159.065,169.700,53.781,160.482
C05312=1007.253,330.957,-159.098,169.708,53.776,160.483
C05313=1007.259,331.205,-159.132,169.716,53.771,160.483
C05314=1007.264,331.453,-159.165,169.724,53.766,160.484
C05315=1007.270,331.701,-159.198,169.732,53.761,160.484
C05316=1007.275,331.948,-159.232,169.739,53.755,160.484
C05317=1007.281,332.196,-159.266,169.747,53.751,160.485
C05318=1007.287,332.443,-159.298,169.755,53.746,160.485
C05319=1007.293,332.691,-159.332,169.762,53.740,160.486
C05320=1007.299,332.938,-159.366,169.770,53.735,160.486
C05321=1007.304,333.186,-159.399,169.779,53.730,160.487
C05322=1007.310,333.434,-159.432,169.786,53.724,160.487
C05323=1007.316,333.682,-159.467,169.794,53.719,160.488
C05324=1007.321,333.929,-159.500,169.802,53.715,160.488
C05325=1007.327,334.177,-159.534,169.809,53.709,160.489
C05326=1007.333,334.425,-159.567,169.817,53.704,160.489
C05327=1007.339,334.672,-159.601,169.825,53.699,160.490
C05328=1007.345,334.920,-159.634,169.833,53.694,160.490
C05329=1007.351,335.168,-159.668,169.841,53.689,160.491
C05330=1007.357,335.415,-159.702,169.849,53.684,160.491
C05331=1007.363,335.663,-159.736,169.857,53.679,160.492
C05332=1007.369,335.910,-159.770,169.865,53.674,160.492
C05333=1007.375,336.159,-159.804,169.873,53.669,160.493
C05334=1007.381,336.406,-159.838,169.881,53.664,160.493
C05335=1007.386,336.654,-159.871,169.889,53.659,160.494
C05336=1007.393,336.901,-159.904,169.898,53.654,160.494
C05337=1007.399,337.149,-159.939,169.905,53.649,160.495
C05338=1007.405,337.396,-159.973,169.913,53.644,160.495
C05339=1007.411,337.643,-160.007,169.921,53.639,160.496
C05340=1007.416,337.892,-160.041,169.929,53.634,160.496
C05341=1007.422,338.140,-160.075,169.938,53.629,160.497
C05342=1007.428,338.387,-160.109,169.946,53.624,160.497
C05343=1007.434,338.634,-160.143,169.954,53.619,160.498
C05344=1007.440,338.882,-160.178,169.962,53.614,160.499
C05345=1007.446,339.098,-160.208,169.968,53.610,160.499
C05346=1007.451,339.314,-160.238,169.976,53.606,160.500
C05347=1007.456,339.531,-160.268,169.983,53.601,160.500
